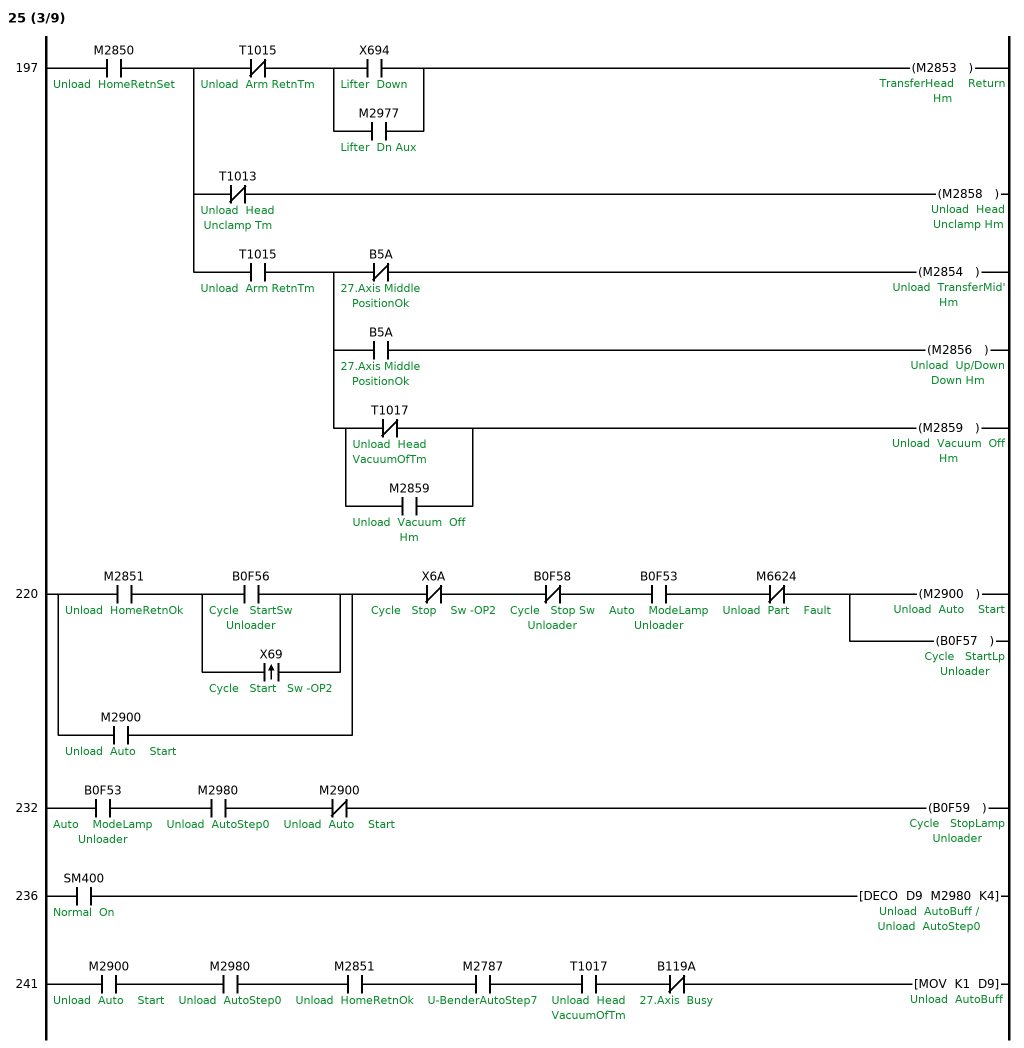
197   LD      M2850  ; Unload  HomeRetnSet
      MPS
      ANI     T1015  ; Unload  Arm RetnTm
      LD      X694  ; Lifter  Down
      OR      M2977  ; Lifter  Dn Aux
      ANB
      OUT     M2853  ; TransferHead    Return  Hm
      MRD
      ANI     T1013  ; Unload  Head    Unclamp Tm
      OUT     M2858  ; Unload  Head    Unclamp Hm
      MPP
      AND     T1015  ; Unload  Arm RetnTm
      MPS
      ANI     B5A  ; 27.Axis Middle  PositionOk
      OUT     M2854  ; Unload  TransferMid' Hm
      MRD
      AND     B5A  ; 27.Axis Middle  PositionOk
      OUT     M2856  ; Unload  Up/Down Down Hm
      MPP
      LDI     T1017  ; Unload  Head    VacuumOfTm
      OR      M2859  ; Unload  Vacuum  Off Hm
      ANB
      OUT     M2859  ; Unload  Vacuum  Off Hm
220   LD      M2851  ; Unload  HomeRetnOk
      LD      B0F56  ; Cycle   StartSw Unloader
      ORP     X69  ; Cycle   Start   Sw -OP2
      ANB
      OR      M2900  ; Unload  Auto    Start
      ANI     X6A  ; Cycle   Stop    Sw -OP2
      ANI     B0F58  ; Cycle   Stop Sw Unloader
      AND     B0F53  ; Auto    ModeLampUnloader
      ANI     M6624  ; Unload  Part    Fault
      OUT     M2900  ; Unload  Auto    Start
      OUT     B0F57  ; Cycle   StartLp Unloader
232   LD      B0F53  ; Auto    ModeLampUnloader
      AND     M2980  ; Unload  AutoStep0
      ANI     M2900  ; Unload  Auto    Start
      OUT     B0F59  ; Cycle   StopLampUnloader
236   LD      SM400  ; Normal  On
      DECO    D9 M2980 K4  ; Unload  AutoBuff
241   LD      M2900  ; Unload  Auto    Start
      AND     M2980  ; Unload  AutoStep0
      AND     M2851  ; Unload  HomeRetnOk
      AND     M2787  ; U-BenderAutoStep7
      AND     T1017  ; Unload  Head    VacuumOfTm
      ANI     B119A  ; 27.Axis  Busy
      MOV     K1 D9
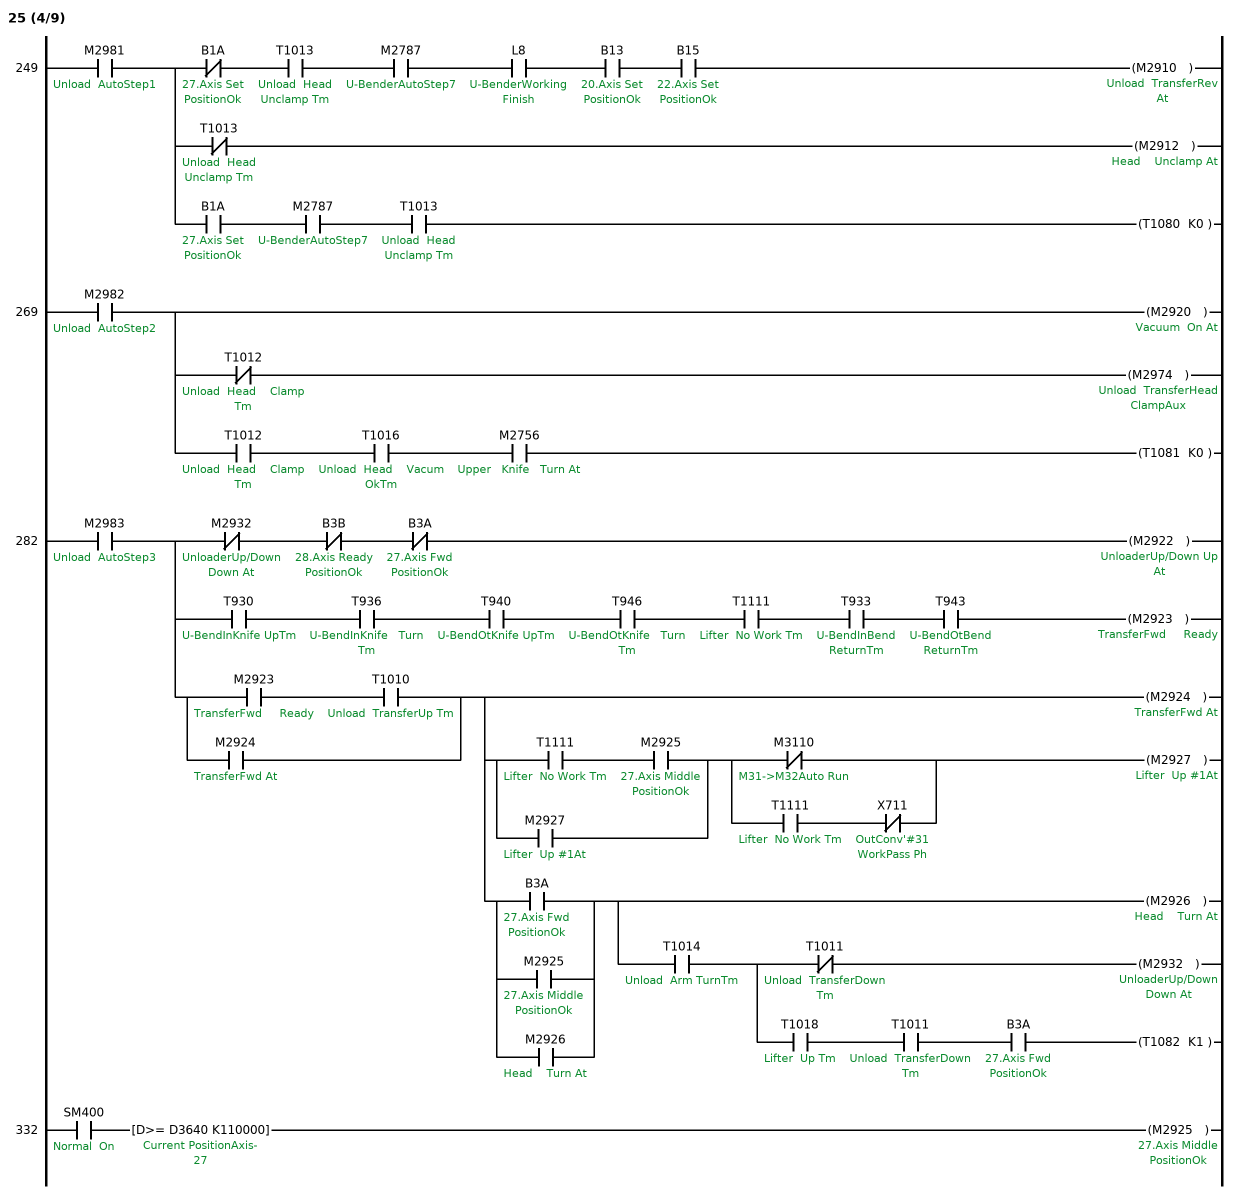
249   LD      M2981  ; Unload  AutoStep1
      MPS
      ANI     B1A  ; 27.Axis Set     PositionOk
      AND     T1013  ; Unload  Head    Unclamp Tm
      AND     M2787  ; U-BenderAutoStep7
      AND     L8  ; U-BenderWorking Finish
      AND     B13  ; 20.Axis Set     PositionOk
      AND     B15  ; 22.Axis Set     PositionOk
      OUT     M2910  ; Unload  TransferRev At
      MRD
      ANI     T1013  ; Unload  Head    Unclamp Tm
      OUT     M2912  ; Head    Unclamp At
      MPP
      AND     B1A  ; 27.Axis Set     PositionOk
      AND     M2787  ; U-BenderAutoStep7
      AND     T1013  ; Unload  Head    Unclamp Tm
      OUT     T1080 K0
269   LD      M2982  ; Unload  AutoStep2
      OUT     M2920  ; Vacuum  On At
      MPS
      ANI     T1012  ; Unload  Head    Clamp Tm
      OUT     M2974  ; Unload  TransferHead    ClampAux
      MPP
      AND     T1012  ; Unload  Head    Clamp Tm
      AND     T1016  ; Unload  Head    Vacum OkTm
      AND     M2756  ; Upper   Knife   Turn At
      OUT     T1081 K0
282   LD      M2983  ; Unload  AutoStep3
      MPS
      ANI     M2932  ; UnloaderUp/Down Down At
      ANI     B3B  ; 28.Axis Ready   PositionOk
      ANI     B3A  ; 27.Axis Fwd     PositionOk
      OUT     M2922  ; UnloaderUp/Down Up At
      MRD
      AND     T930  ; U-BendInKnife UpTm
      AND     T936  ; U-BendInKnife   Turn Tm
      AND     T940  ; U-BendOtKnife UpTm
      AND     T946  ; U-BendOtKnife   Turn Tm
      AND     T1111  ; Lifter  No Work Tm
      AND     T933  ; U-BendInBend    ReturnTm
      AND     T943  ; U-BendOtBend    ReturnTm
      OUT     M2923  ; TransferFwd     Ready
      MPP
      LD      M2923  ; TransferFwd     Ready
      AND     T1010  ; Unload  TransferUp Tm
      OR      M2924  ; TransferFwd At
      ANB
      OUT     M2924  ; TransferFwd At
      MPS
      LD      T1111  ; Lifter  No Work Tm
      AND     M2925  ; 27.Axis Middle  PositionOk
      OR      M2927  ; Lifter  Up #1At
      ANB
      LDI     M3110  ; M31->M32Auto Run
      LD      T1111  ; Lifter  No Work Tm
      ANI     X711  ; OutConv'#31 WorkPass Ph
      ORB
      ANB
      OUT     M2927  ; Lifter  Up #1At
      MPP
      LD      B3A  ; 27.Axis Fwd     PositionOk
      OR      M2925  ; 27.Axis Middle  PositionOk
      OR      M2926  ; Head    Turn At
      ANB
      OUT     M2926  ; Head    Turn At
      AND     T1014  ; Unload  Arm TurnTm
      MPS
      ANI     T1011  ; Unload  TransferDown Tm
      OUT     M2932  ; UnloaderUp/Down Down At
      MPP
      AND     T1018  ; Lifter  Up Tm
      AND     T1011  ; Unload  TransferDown Tm
      AND     B3A  ; 27.Axis Fwd     PositionOk
      OUT     T1082 K1
332   LD      SM400  ; Normal  On
      ANDD>=  D3640 K110000  ; Current PositionAxis-27
      OUT     M2925  ; 27.Axis Middle  PositionOk
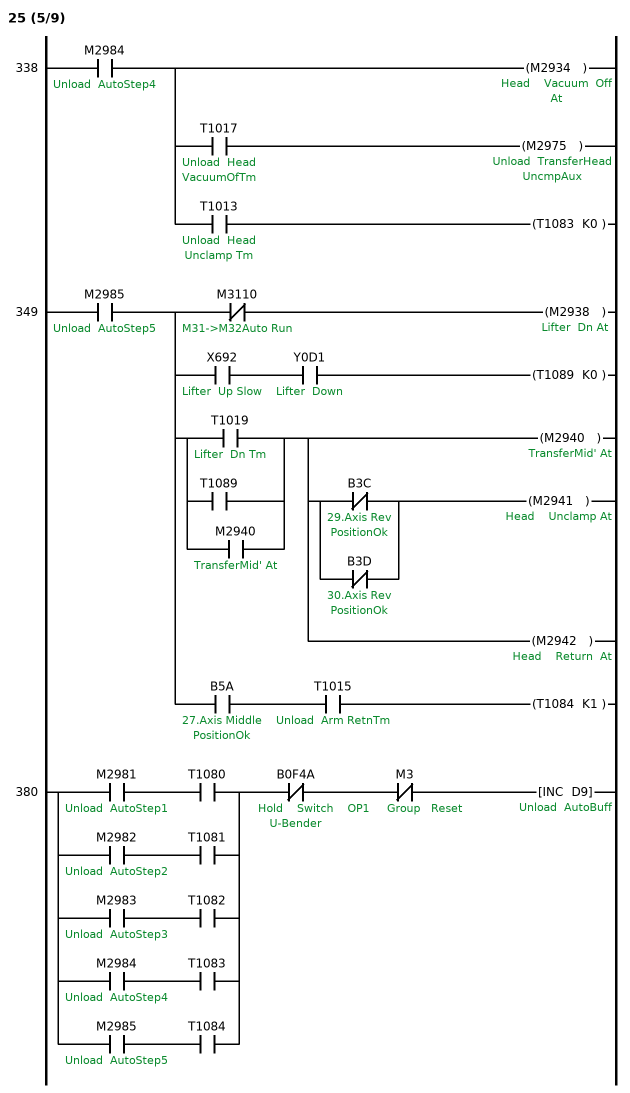
338   LD      M2984  ; Unload  AutoStep4
      OUT     M2934  ; Head    Vacuum  Off At
      MPS
      AND     T1017  ; Unload  Head    VacuumOfTm
      OUT     M2975  ; Unload  TransferHead    UncmpAux
      MPP
      AND     T1013  ; Unload  Head    Unclamp Tm
      OUT     T1083 K0
349   LD      M2985  ; Unload  AutoStep5
      MPS
      ANI     M3110  ; M31->M32Auto Run
      OUT     M2938  ; Lifter  Dn At
      MRD
      AND     X692  ; Lifter  Up Slow
      AND     Y0D1  ; Lifter  Down
      OUT     T1089 K0
      MRD
      LD      T1019  ; Lifter  Dn Tm
      OR      T1089
      OR      M2940  ; TransferMid' At
      ANB
      OUT     M2940  ; TransferMid' At
      MPS
      LDI     B3C  ; 29.Axis Rev     PositionOk
      ORI     B3D  ; 30.Axis Rev     PositionOk
      ANB
      OUT     M2941  ; Head    Unclamp At
      MPP
      OUT     M2942  ; Head    Return  At
      MPP
      AND     B5A  ; 27.Axis Middle  PositionOk
      AND     T1015  ; Unload  Arm RetnTm
      OUT     T1084 K1
380   LD      M2981  ; Unload  AutoStep1
      AND     T1080
      LD      M2982  ; Unload  AutoStep2
      AND     T1081
      ORB
      LD      M2983  ; Unload  AutoStep3
      AND     T1082
      ORB
      LD      M2984  ; Unload  AutoStep4
      AND     T1083
      ORB
      LD      M2985  ; Unload  AutoStep5
      AND     T1084
      ORB
      ANI     B0F4A  ; Hold    Switch  U-Bender
      ANI     M3  ; OP1     Group   Reset
      INC     D9
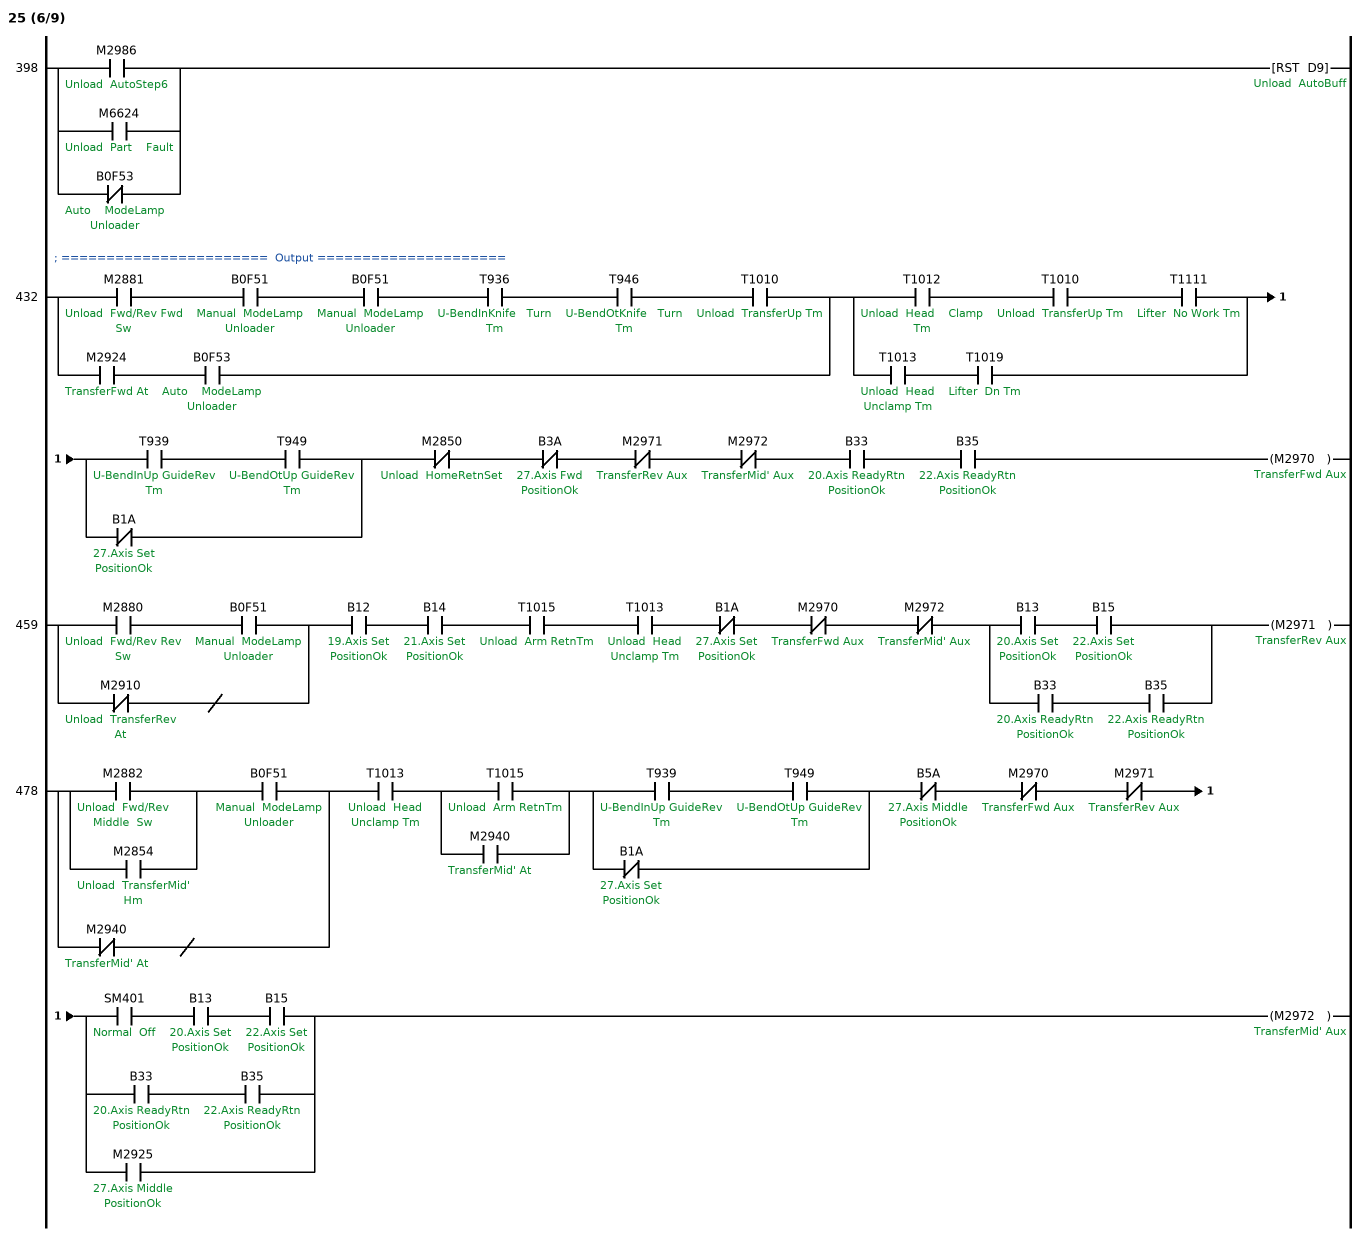
398   LD      M2986  ; Unload  AutoStep6
      OR      M6624  ; Unload  Part    Fault
      ORI     B0F53  ; Auto    ModeLampUnloader
      RST     D9  ; Unload  AutoBuff
; =======================  Output =====================
432   LD      M2881  ; Unload  Fwd/Rev Fwd Sw
      AND     B0F51  ; Manual  ModeLampUnloader
      AND     B0F51  ; Manual  ModeLampUnloader
      AND     T936  ; U-BendInKnife   Turn Tm
      AND     T946  ; U-BendOtKnife   Turn Tm
      AND     T1010  ; Unload  TransferUp Tm
      LD      M2924  ; TransferFwd At
      AND     B0F53  ; Auto    ModeLampUnloader
      ORB
      LD      T1012  ; Unload  Head    Clamp Tm
      AND     T1010  ; Unload  TransferUp Tm
      AND     T1111  ; Lifter  No Work Tm
      LD      T1013  ; Unload  Head    Unclamp Tm
      AND     T1019  ; Lifter  Dn Tm
      ORB
      ANB
      LD      T939  ; U-BendInUp GuideRev Tm
      AND     T949  ; U-BendOtUp GuideRev Tm
      ORI     B1A  ; 27.Axis Set     PositionOk
      ANB
      ANI     M2850  ; Unload  HomeRetnSet
      ANI     B3A  ; 27.Axis Fwd     PositionOk
      ANI     M2971  ; TransferRev Aux
      ANI     M2972  ; TransferMid' Aux
      AND     B33  ; 20.Axis ReadyRtnPositionOk
      AND     B35  ; 22.Axis ReadyRtnPositionOk
      OUT     M2970  ; TransferFwd Aux
459   LD      M2880  ; Unload  Fwd/Rev Rev Sw
      AND     B0F51  ; Manual  ModeLampUnloader
      LDI     M2910  ; Unload  TransferRev At
      INV
      ORB
      AND     B12  ; 19.Axis Set     PositionOk
      AND     B14  ; 21.Axis Set     PositionOk
      AND     T1015  ; Unload  Arm RetnTm
      AND     T1013  ; Unload  Head    Unclamp Tm
      ANI     B1A  ; 27.Axis Set     PositionOk
      ANI     M2970  ; TransferFwd Aux
      ANI     M2972  ; TransferMid' Aux
      LD      B13  ; 20.Axis Set     PositionOk
      AND     B15  ; 22.Axis Set     PositionOk
      LD      B33  ; 20.Axis ReadyRtnPositionOk
      AND     B35  ; 22.Axis ReadyRtnPositionOk
      ORB
      ANB
      OUT     M2971  ; TransferRev Aux
478   LD      M2882  ; Unload  Fwd/Rev Middle  Sw
      OR      M2854  ; Unload  TransferMid' Hm
      AND     B0F51  ; Manual  ModeLampUnloader
      LDI     M2940  ; TransferMid' At
      INV
      ORB
      AND     T1013  ; Unload  Head    Unclamp Tm
      LD      T1015  ; Unload  Arm RetnTm
      OR      M2940  ; TransferMid' At
      ANB
      LD      T939  ; U-BendInUp GuideRev Tm
      AND     T949  ; U-BendOtUp GuideRev Tm
      ORI     B1A  ; 27.Axis Set     PositionOk
      ANB
      ANI     B5A  ; 27.Axis Middle  PositionOk
      ANI     M2970  ; TransferFwd Aux
      ANI     M2971  ; TransferRev Aux
      LD      SM401  ; Normal  Off
      AND     B13  ; 20.Axis Set     PositionOk
      AND     B15  ; 22.Axis Set     PositionOk
      LD      B33  ; 20.Axis ReadyRtnPositionOk
      AND     B35  ; 22.Axis ReadyRtnPositionOk
      ORB
      OR      M2925  ; 27.Axis Middle  PositionOk
      ANB
      OUT     M2972  ; TransferMid' Aux
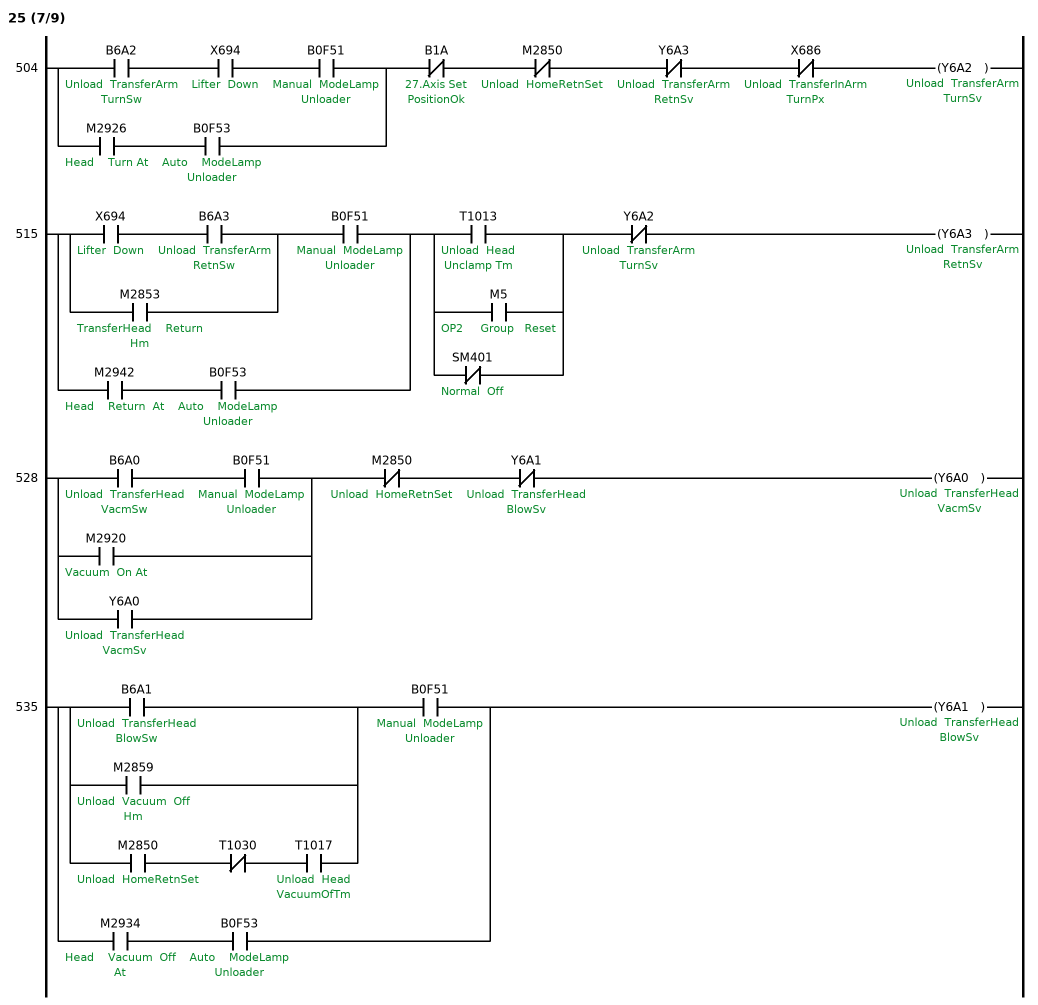
504   LD      B6A2  ; Unload  TransferArm TurnSw
      AND     X694  ; Lifter  Down
      AND     B0F51  ; Manual  ModeLampUnloader
      LD      M2926  ; Head    Turn At
      AND     B0F53  ; Auto    ModeLampUnloader
      ORB
      ANI     B1A  ; 27.Axis Set     PositionOk
      ANI     M2850  ; Unload  HomeRetnSet
      ANI     Y6A3  ; Unload  TransferArm RetnSv
      ANI     X686  ; Unload  TransferInArm   TurnPx
      OUT     Y6A2  ; Unload  TransferArm TurnSv
515   LD      X694  ; Lifter  Down
      AND     B6A3  ; Unload  TransferArm RetnSw
      OR      M2853  ; TransferHead    Return  Hm
      AND     B0F51  ; Manual  ModeLampUnloader
      LD      M2942  ; Head    Return  At
      AND     B0F53  ; Auto    ModeLampUnloader
      ORB
      LD      T1013  ; Unload  Head    Unclamp Tm
      OR      M5  ; OP2     Group   Reset
      ORI     SM401  ; Normal  Off
      ANB
      ANI     Y6A2  ; Unload  TransferArm TurnSv
      OUT     Y6A3  ; Unload  TransferArm RetnSv
528   LD      B6A0  ; Unload  TransferHeadVacmSw
      AND     B0F51  ; Manual  ModeLampUnloader
      OR      M2920  ; Vacuum  On At
      OR      Y6A0  ; Unload  TransferHeadVacmSv
      ANI     M2850  ; Unload  HomeRetnSet
      ANI     Y6A1  ; Unload  TransferHeadBlowSv
      OUT     Y6A0  ; Unload  TransferHeadVacmSv
535   LD      B6A1  ; Unload  TransferHeadBlowSw
      OR      M2859  ; Unload  Vacuum  Off Hm
      LD      M2850  ; Unload  HomeRetnSet
      ANI     T1030
      AND     T1017  ; Unload  Head    VacuumOfTm
      ORB
      AND     B0F51  ; Manual  ModeLampUnloader
      LD      M2934  ; Head    Vacuum  Off At
      AND     B0F53  ; Auto    ModeLampUnloader
      ORB
      OUT     Y6A1  ; Unload  TransferHeadBlowSv
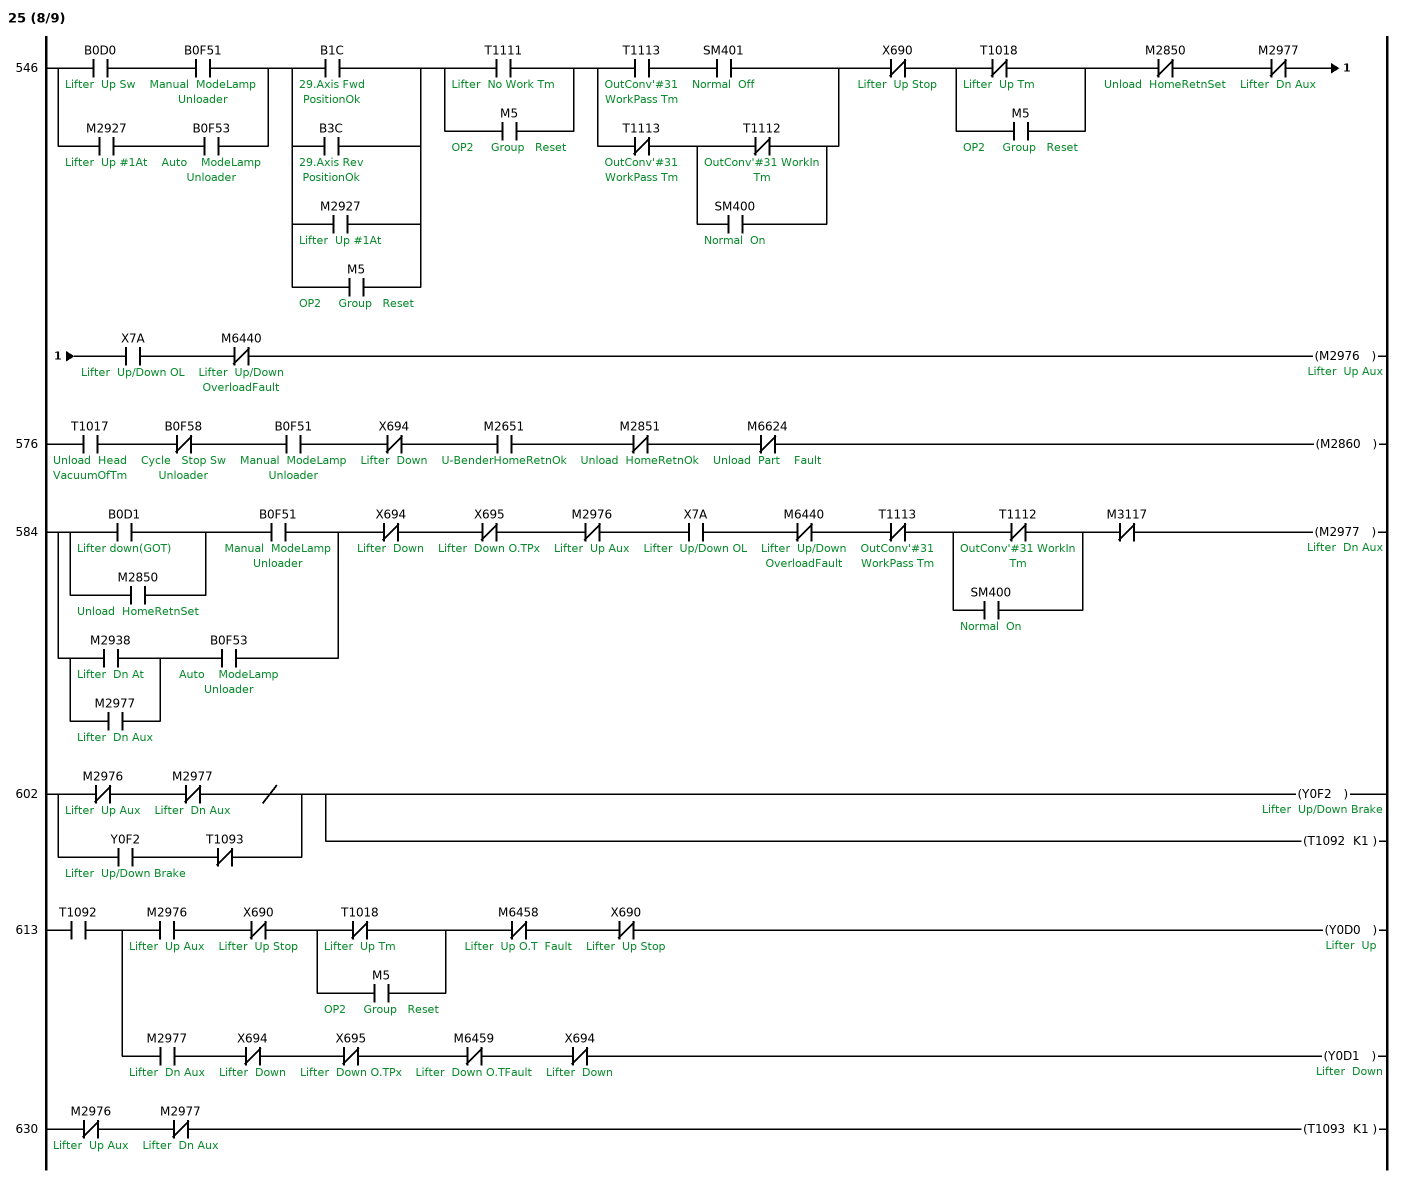
546   LD      B0D0  ; Lifter  Up Sw
      AND     B0F51  ; Manual  ModeLampUnloader
      LD      M2927  ; Lifter  Up #1At
      AND     B0F53  ; Auto    ModeLampUnloader
      ORB
      LD      B1C  ; 29.Axis Fwd     PositionOk
      OR      B3C  ; 29.Axis Rev     PositionOk
      OR      M2927  ; Lifter  Up #1At
      OR      M5  ; OP2     Group   Reset
      ANB
      LD      T1111  ; Lifter  No Work Tm
      OR      M5  ; OP2     Group   Reset
      ANB
      LD      T1113  ; OutConv'#31 WorkPass Tm
      AND     SM401  ; Normal  Off
      LDI     T1113  ; OutConv'#31 WorkPass Tm
      LDI     T1112  ; OutConv'#31 WorkIn  Tm
      OR      SM400  ; Normal  On
      ANB
      ORB
      ANB
      ANI     X690  ; Lifter  Up Stop
      LDI     T1018  ; Lifter  Up Tm
      OR      M5  ; OP2     Group   Reset
      ANB
      ANI     M2850  ; Unload  HomeRetnSet
      ANI     M2977  ; Lifter  Dn Aux
      AND     X7A  ; Lifter  Up/Down OL
      ANI     M6440  ; Lifter  Up/Down OverloadFault
      OUT     M2976  ; Lifter  Up Aux
576   LD      T1017  ; Unload  Head    VacuumOfTm
      ANI     B0F58  ; Cycle   Stop Sw Unloader
      AND     B0F51  ; Manual  ModeLampUnloader
      ANI     X694  ; Lifter  Down
      AND     M2651  ; U-BenderHomeRetnOk
      ANI     M2851  ; Unload  HomeRetnOk
      ANI     M6624  ; Unload  Part    Fault
      OUT     M2860
584   LD      B0D1  ; Lifter down(GOT)
      OR      M2850  ; Unload  HomeRetnSet
      AND     B0F51  ; Manual  ModeLampUnloader
      LD      M2938  ; Lifter  Dn At
      OR      M2977  ; Lifter  Dn Aux
      AND     B0F53  ; Auto    ModeLampUnloader
      ORB
      ANI     X694  ; Lifter  Down
      ANI     X695  ; Lifter  Down O.TPx
      ANI     M2976  ; Lifter  Up Aux
      AND     X7A  ; Lifter  Up/Down OL
      ANI     M6440  ; Lifter  Up/Down OverloadFault
      ANI     T1113  ; OutConv'#31 WorkPass Tm
      LDI     T1112  ; OutConv'#31 WorkIn  Tm
      OR      SM400  ; Normal  On
      ANB
      ANI     M3117
      OUT     M2977  ; Lifter  Dn Aux
602   LDI     M2976  ; Lifter  Up Aux
      ANI     M2977  ; Lifter  Dn Aux
      INV
      LD      Y0F2  ; Lifter  Up/Down Brake
      ANI     T1093
      ORB
      OUT     Y0F2  ; Lifter  Up/Down Brake
      OUT     T1092 K1
613   LD      T1092
      MPS
      AND     M2976  ; Lifter  Up Aux
      ANI     X690  ; Lifter  Up Stop
      LDI     T1018  ; Lifter  Up Tm
      OR      M5  ; OP2     Group   Reset
      ANB
      ANI     M6458  ; Lifter  Up O.T  Fault
      ANI     X690  ; Lifter  Up Stop
      OUT     Y0D0  ; Lifter  Up
      MPP
      AND     M2977  ; Lifter  Dn Aux
      ANI     X694  ; Lifter  Down
      ANI     X695  ; Lifter  Down O.TPx
      ANI     M6459  ; Lifter  Down O.TFault
      ANI     X694  ; Lifter  Down
      OUT     Y0D1  ; Lifter  Down
630   LDI     M2976  ; Lifter  Up Aux
      ANI     M2977  ; Lifter  Dn Aux
      OUT     T1093 K1
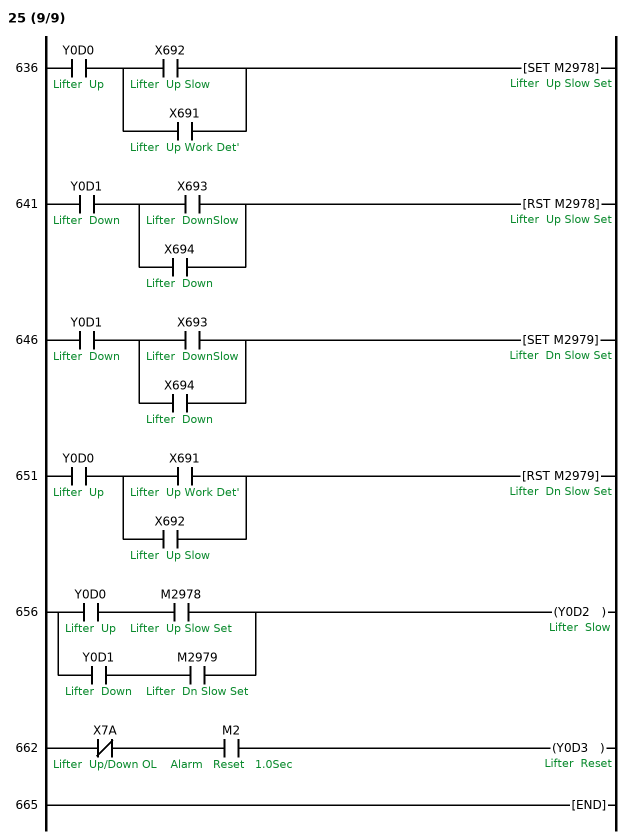
636   LD      Y0D0  ; Lifter  Up
      LD      X692  ; Lifter  Up Slow
      OR      X691  ; Lifter  Up Work Det'
      ANB
      SET     M2978  ; Lifter  Up Slow Set
641   LD      Y0D1  ; Lifter  Down
      LD      X693  ; Lifter  DownSlow
      OR      X694  ; Lifter  Down
      ANB
      RST     M2978  ; Lifter  Up Slow Set
646   LD      Y0D1  ; Lifter  Down
      LD      X693  ; Lifter  DownSlow
      OR      X694  ; Lifter  Down
      ANB
      SET     M2979  ; Lifter  Dn Slow Set
651   LD      Y0D0  ; Lifter  Up
      LD      X691  ; Lifter  Up Work Det'
      OR      X692  ; Lifter  Up Slow
      ANB
      RST     M2979  ; Lifter  Dn Slow Set
656   LD      Y0D0  ; Lifter  Up
      AND     M2978  ; Lifter  Up Slow Set
      LD      Y0D1  ; Lifter  Down
      AND     M2979  ; Lifter  Dn Slow Set
      ORB
      OUT     Y0D2  ; Lifter  Slow
662   LDI     X7A  ; Lifter  Up/Down OL
      AND     M2  ; Alarm   Reset   1.0Sec
      OUT     Y0D3  ; Lifter  Reset
665   END
END_PROGRAM

PROGRAM 26  // Out Conveyor
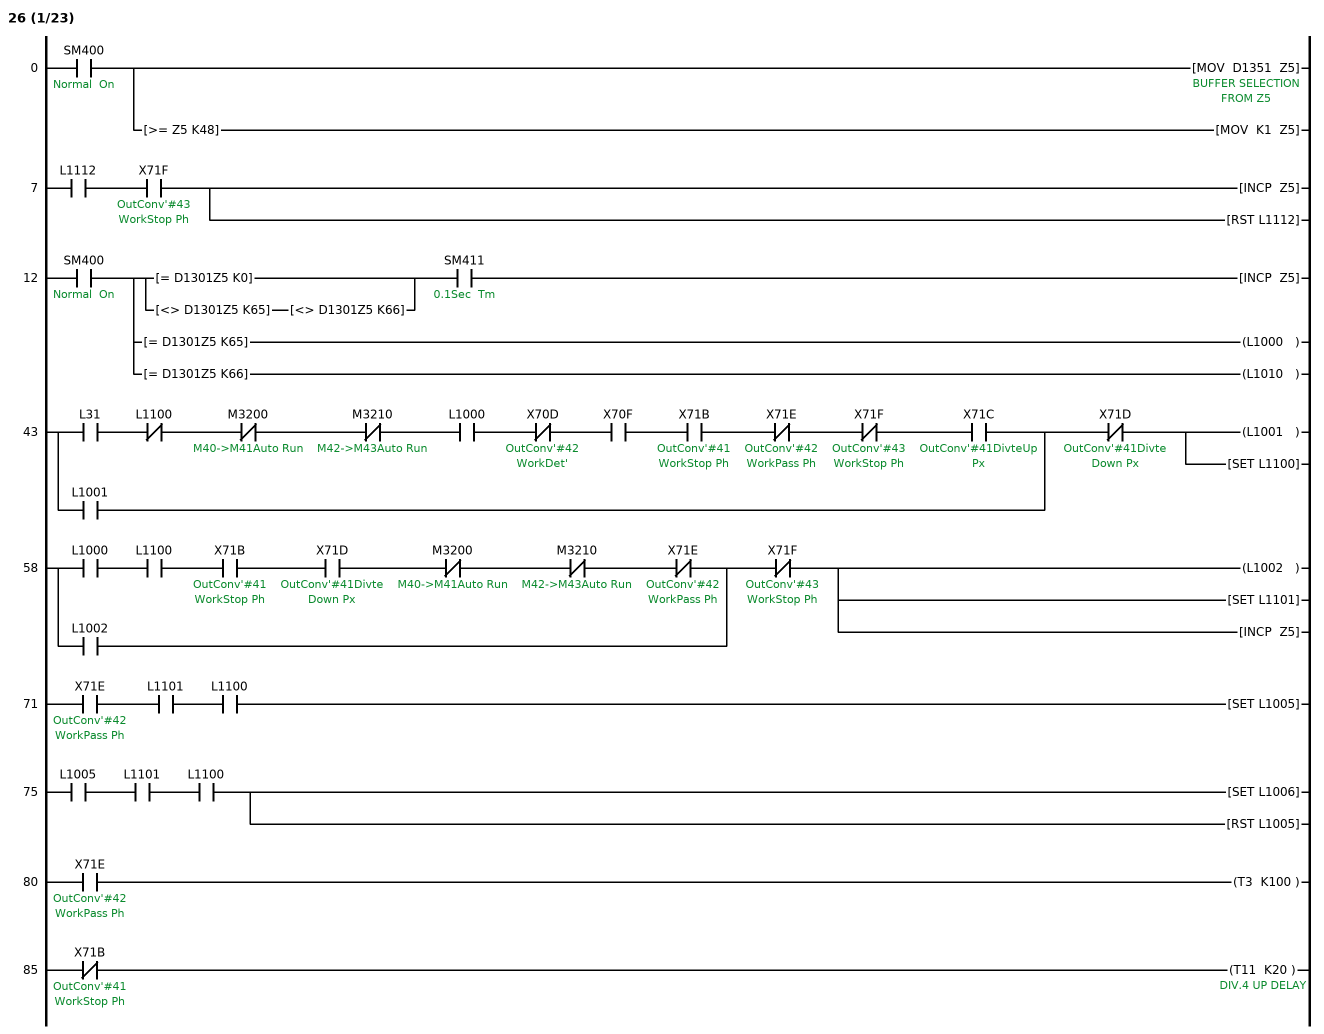
0     LD      SM400  ; Normal  On
      MOV     D1351 Z5  ; BUFFER SELECTION FROM Z5
      AND>=   Z5 K48
      MOV     K1 Z5
7     LD      L1112
      AND     X71F  ; OutConv'#43 WorkStop Ph
      INCP    Z5
      RST     L1112
12    LD      SM400  ; Normal  On
      MPS
      LD=     D1301Z5 K0
      LD<>    D1301Z5 K65
      AND<>   D1301Z5 K66
      ORB
      ANB
      AND     SM411  ; 0.1Sec  Tm
      INCP    Z5
      MRD
      AND=    D1301Z5 K65
      OUT     L1000
      MPP
      AND=    D1301Z5 K66
      OUT     L1010
43    LD      L31
      ANI     L1100
      ANI     M3200  ; M40->M41Auto Run
      ANI     M3210  ; M42->M43Auto Run
      AND     L1000
      ANI     X70D  ; OutConv'#42 WorkDet'
      AND     X70F
      AND     X71B  ; OutConv'#41 WorkStop Ph
      ANI     X71E  ; OutConv'#42 WorkPass Ph
      ANI     X71F  ; OutConv'#43 WorkStop Ph
      AND     X71C  ; OutConv'#41DivteUp Px
      OR      L1001
      ANI     X71D  ; OutConv'#41DivteDown Px
      OUT     L1001
      SET     L1100
58    LD      L1000
      AND     L1100
      AND     X71B  ; OutConv'#41 WorkStop Ph
      AND     X71D  ; OutConv'#41DivteDown Px
      ANI     M3200  ; M40->M41Auto Run
      ANI     M3210  ; M42->M43Auto Run
      ANI     X71E  ; OutConv'#42 WorkPass Ph
      OR      L1002
      ANI     X71F  ; OutConv'#43 WorkStop Ph
      OUT     L1002
      SET     L1101
      INCP    Z5
71    LD      X71E  ; OutConv'#42 WorkPass Ph
      AND     L1101
      AND     L1100
      SET     L1005
75    LD      L1005
      AND     L1101
      AND     L1100
      SET     L1006
      RST     L1005
80    LD      X71E  ; OutConv'#42 WorkPass Ph
      OUT     T3 K100
85    LDI     X71B  ; OutConv'#41 WorkStop Ph
      OUT     T11 K20  ; DIV.4 UP DELAY
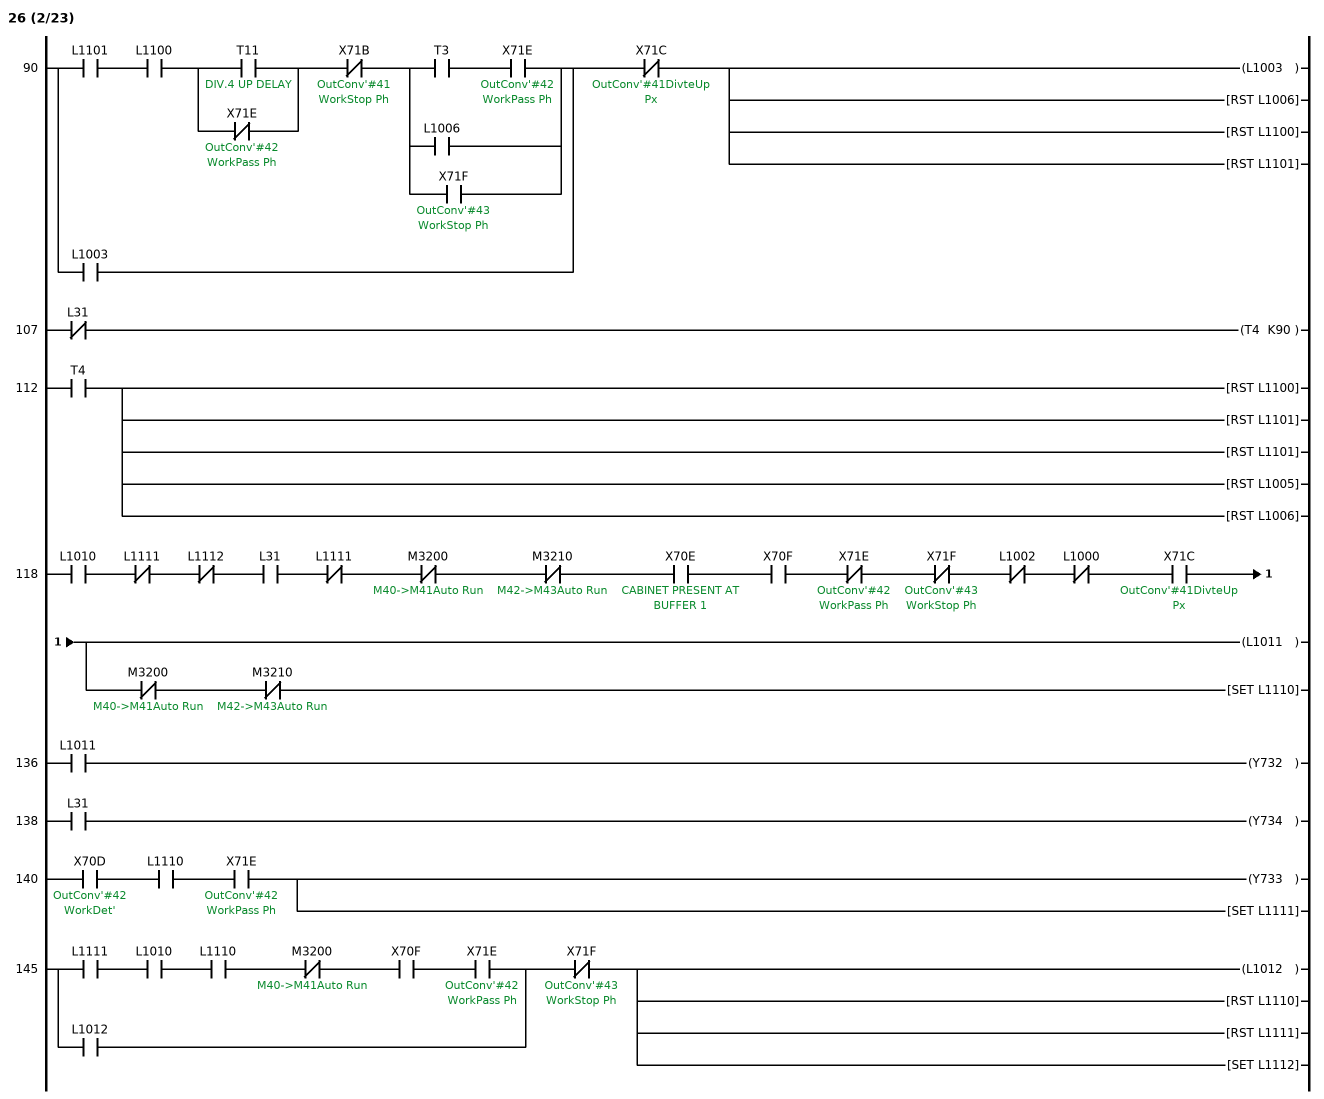
90    LD      L1101
      AND     L1100
      LD      T11  ; DIV.4 UP DELAY
      ORI     X71E  ; OutConv'#42 WorkPass Ph
      ANB
      ANI     X71B  ; OutConv'#41 WorkStop Ph
      LD      T3
      AND     X71E  ; OutConv'#42 WorkPass Ph
      OR      L1006
      OR      X71F  ; OutConv'#43 WorkStop Ph
      ANB
      OR      L1003
      ANI     X71C  ; OutConv'#41DivteUp Px
      OUT     L1003
      RST     L1006
      RST     L1100
      RST     L1101
107   LDI     L31
      OUT     T4 K90
112   LD      T4
      RST     L1100
      RST     L1101
      RST     L1101
      RST     L1005
      RST     L1006
118   LD      L1010
      ANI     L1111
      ANI     L1112
      AND     L31
      ANI     L1111
      ANI     M3200  ; M40->M41Auto Run
      ANI     M3210  ; M42->M43Auto Run
      AND     X70E  ; CABINET PRESENT AT BUFFER 1
      AND     X70F
      ANI     X71E  ; OutConv'#42 WorkPass Ph
      ANI     X71F  ; OutConv'#43 WorkStop Ph
      ANI     L1002
      ANI     L1000
      AND     X71C  ; OutConv'#41DivteUp Px
      OUT     L1011
      ANI     M3200  ; M40->M41Auto Run
      ANI     M3210  ; M42->M43Auto Run
      SET     L1110
136   LD      L1011
      OUT     Y732
138   LD      L31
      OUT     Y734
140   LD      X70D  ; OutConv'#42 WorkDet'
      AND     L1110
      AND     X71E  ; OutConv'#42 WorkPass Ph
      OUT     Y733
      SET     L1111
145   LD      L1111
      AND     L1010
      AND     L1110
      ANI     M3200  ; M40->M41Auto Run
      AND     X70F
      AND     X71E  ; OutConv'#42 WorkPass Ph
      OR      L1012
      ANI     X71F  ; OutConv'#43 WorkStop Ph
      OUT     L1012
      RST     L1110
      RST     L1111
      SET     L1112
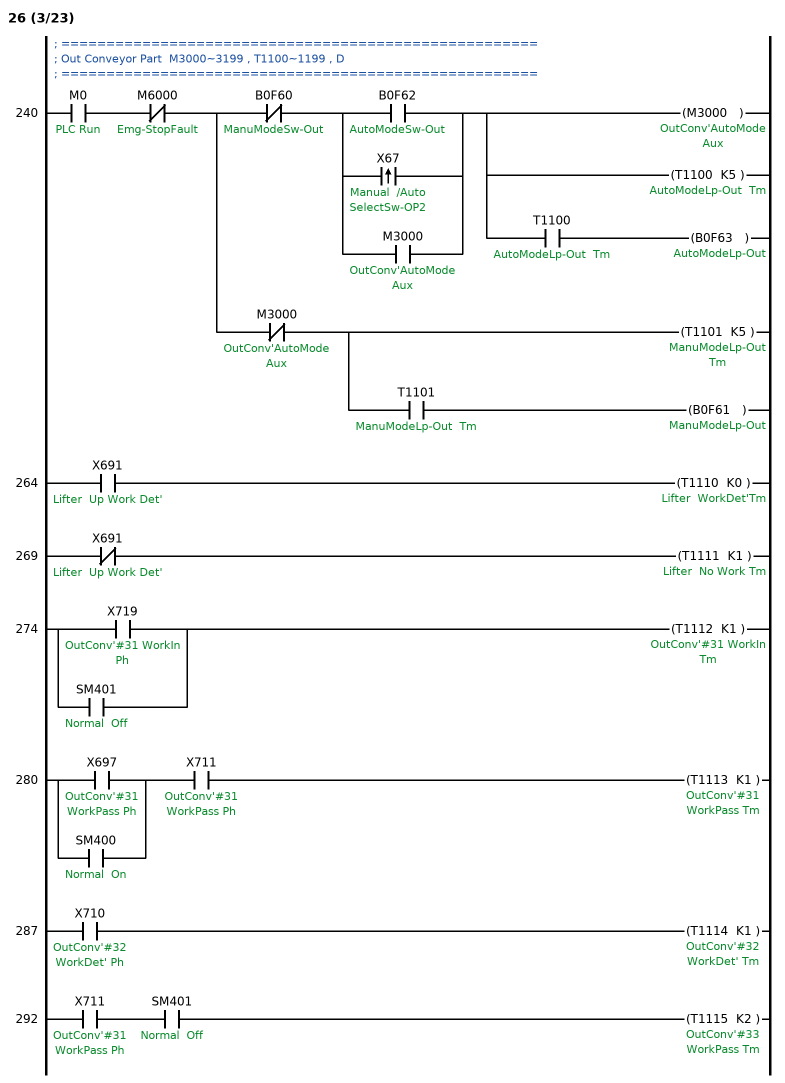
; =====================================================
; Out Conveyor Part  M3000~3199 , T1100~1199 , D
; =====================================================
240   LD      M0  ; PLC Run
      ANI     M6000  ; Emg-StopFault
      MPS
      ANI     B0F60  ; ManuModeSw-Out
      LD      B0F62  ; AutoModeSw-Out
      ORP     X67  ; Manual  /Auto   SelectSw-OP2
      OR      M3000  ; OutConv'AutoModeAux
      ANB
      OUT     M3000  ; OutConv'AutoModeAux
      OUT     T1100 K5  ; AutoModeLp-Out  Tm
      AND     T1100  ; AutoModeLp-Out  Tm
      OUT     B0F63  ; AutoModeLp-Out
      MPP
      ANI     M3000  ; OutConv'AutoModeAux
      OUT     T1101 K5  ; ManuModeLp-Out  Tm
      AND     T1101  ; ManuModeLp-Out  Tm
      OUT     B0F61  ; ManuModeLp-Out
264   LD      X691  ; Lifter  Up Work Det'
      OUT     T1110 K0  ; Lifter  WorkDet'Tm
269   LDI     X691  ; Lifter  Up Work Det'
      OUT     T1111 K1  ; Lifter  No Work Tm
274   LD      X719  ; OutConv'#31 WorkIn  Ph
      OR      SM401  ; Normal  Off
      OUT     T1112 K1  ; OutConv'#31 WorkIn  Tm
280   LD      X697  ; OutConv'#31 WorkPass Ph
      OR      SM400  ; Normal  On
      AND     X711  ; OutConv'#31 WorkPass Ph
      OUT     T1113 K1  ; OutConv'#31 WorkPass Tm
287   LD      X710  ; OutConv'#32 WorkDet' Ph
      OUT     T1114 K1  ; OutConv'#32 WorkDet' Tm
292   LD      X711  ; OutConv'#31 WorkPass Ph
      AND     SM401  ; Normal  Off
      OUT     T1115 K2  ; OutConv'#33 WorkPass Tm
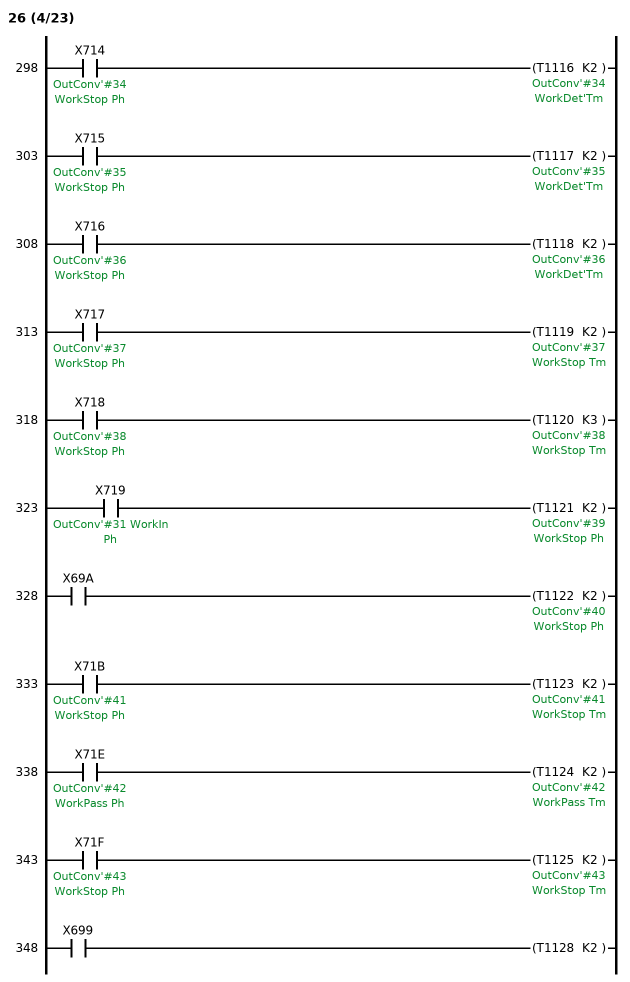
298   LD      X714  ; OutConv'#34 WorkStop Ph
      OUT     T1116 K2  ; OutConv'#34 WorkDet'Tm
303   LD      X715  ; OutConv'#35 WorkStop Ph
      OUT     T1117 K2  ; OutConv'#35 WorkDet'Tm
308   LD      X716  ; OutConv'#36 WorkStop Ph
      OUT     T1118 K2  ; OutConv'#36 WorkDet'Tm
313   LD      X717  ; OutConv'#37 WorkStop Ph
      OUT     T1119 K2  ; OutConv'#37 WorkStop Tm
318   LD      X718  ; OutConv'#38 WorkStop Ph
      OUT     T1120 K3  ; OutConv'#38 WorkStop Tm
323   LD      X719  ; OutConv'#31 WorkIn  Ph
      OUT     T1121 K2  ; OutConv'#39 WorkStop Ph
328   LD      X69A
      OUT     T1122 K2  ; OutConv'#40 WorkStop Ph
333   LD      X71B  ; OutConv'#41 WorkStop Ph
      OUT     T1123 K2  ; OutConv'#41 WorkStop Tm
338   LD      X71E  ; OutConv'#42 WorkPass Ph
      OUT     T1124 K2  ; OutConv'#42 WorkPass Tm
343   LD      X71F  ; OutConv'#43 WorkStop Ph
      OUT     T1125 K2  ; OutConv'#43 WorkStop Tm
348   LD      X699
      OUT     T1128 K2
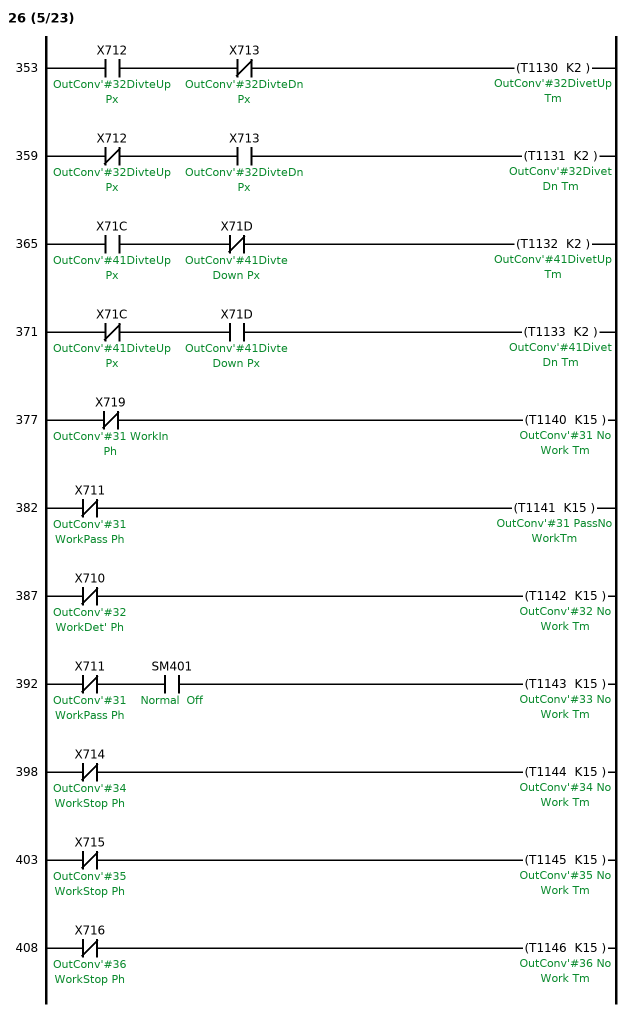
353   LD      X712  ; OutConv'#32DivteUp Px
      ANI     X713  ; OutConv'#32DivteDn Px
      OUT     T1130 K2  ; OutConv'#32DivetUp Tm
359   LDI     X712  ; OutConv'#32DivteUp Px
      AND     X713  ; OutConv'#32DivteDn Px
      OUT     T1131 K2  ; OutConv'#32DivetDn Tm
365   LD      X71C  ; OutConv'#41DivteUp Px
      ANI     X71D  ; OutConv'#41DivteDown Px
      OUT     T1132 K2  ; OutConv'#41DivetUp Tm
371   LDI     X71C  ; OutConv'#41DivteUp Px
      AND     X71D  ; OutConv'#41DivteDown Px
      OUT     T1133 K2  ; OutConv'#41DivetDn Tm
377   LDI     X719  ; OutConv'#31 WorkIn  Ph
      OUT     T1140 K15  ; OutConv'#31 No  Work Tm
382   LDI     X711  ; OutConv'#31 WorkPass Ph
      OUT     T1141 K15  ; OutConv'#31 PassNo  WorkTm
387   LDI     X710  ; OutConv'#32 WorkDet' Ph
      OUT     T1142 K15  ; OutConv'#32 No  Work Tm
392   LDI     X711  ; OutConv'#31 WorkPass Ph
      AND     SM401  ; Normal  Off
      OUT     T1143 K15  ; OutConv'#33 No  Work Tm
398   LDI     X714  ; OutConv'#34 WorkStop Ph
      OUT     T1144 K15  ; OutConv'#34 No  Work Tm
403   LDI     X715  ; OutConv'#35 WorkStop Ph
      OUT     T1145 K15  ; OutConv'#35 No  Work Tm
408   LDI     X716  ; OutConv'#36 WorkStop Ph
      OUT     T1146 K15  ; OutConv'#36 No  Work Tm
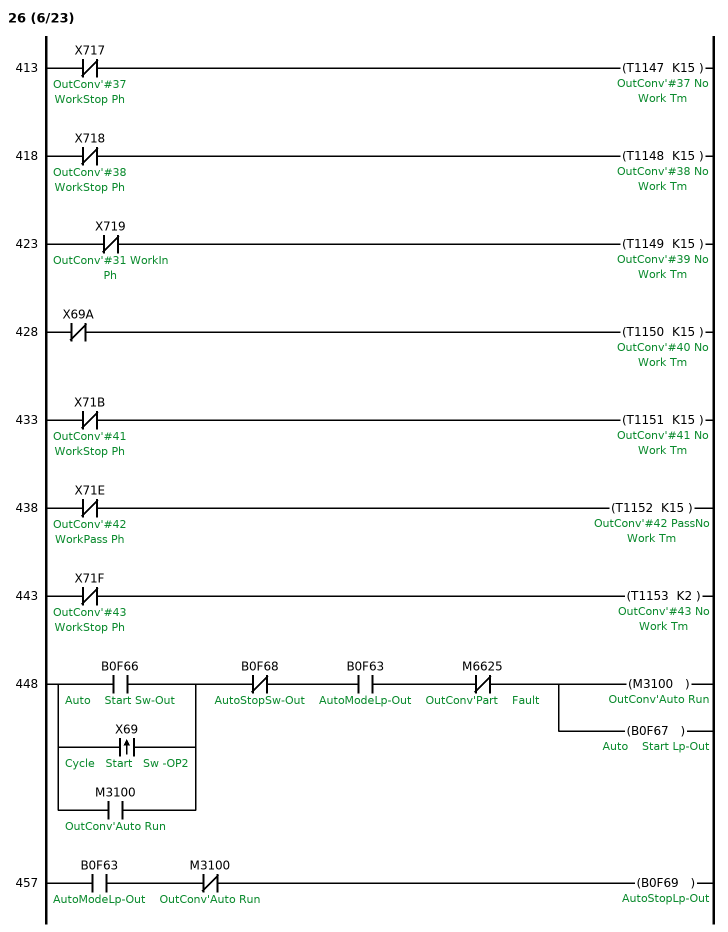
413   LDI     X717  ; OutConv'#37 WorkStop Ph
      OUT     T1147 K15  ; OutConv'#37 No  Work Tm
418   LDI     X718  ; OutConv'#38 WorkStop Ph
      OUT     T1148 K15  ; OutConv'#38 No  Work Tm
423   LDI     X719  ; OutConv'#31 WorkIn  Ph
      OUT     T1149 K15  ; OutConv'#39 No  Work Tm
428   LDI     X69A
      OUT     T1150 K15  ; OutConv'#40 No  Work Tm
433   LDI     X71B  ; OutConv'#41 WorkStop Ph
      OUT     T1151 K15  ; OutConv'#41 No  Work Tm
438   LDI     X71E  ; OutConv'#42 WorkPass Ph
      OUT     T1152 K15  ; OutConv'#42 PassNo Work Tm
443   LDI     X71F  ; OutConv'#43 WorkStop Ph
      OUT     T1153 K2  ; OutConv'#43 No  Work Tm
448   LD      B0F66  ; Auto    Start Sw-Out
      ORP     X69  ; Cycle   Start   Sw -OP2
      OR      M3100  ; OutConv'Auto Run
      ANI     B0F68  ; AutoStopSw-Out
      AND     B0F63  ; AutoModeLp-Out
      ANI     M6625  ; OutConv'Part    Fault
      OUT     M3100  ; OutConv'Auto Run
      OUT     B0F67  ; Auto    Start Lp-Out
457   LD      B0F63  ; AutoModeLp-Out
      ANI     M3100  ; OutConv'Auto Run
      OUT     B0F69  ; AutoStopLp-Out
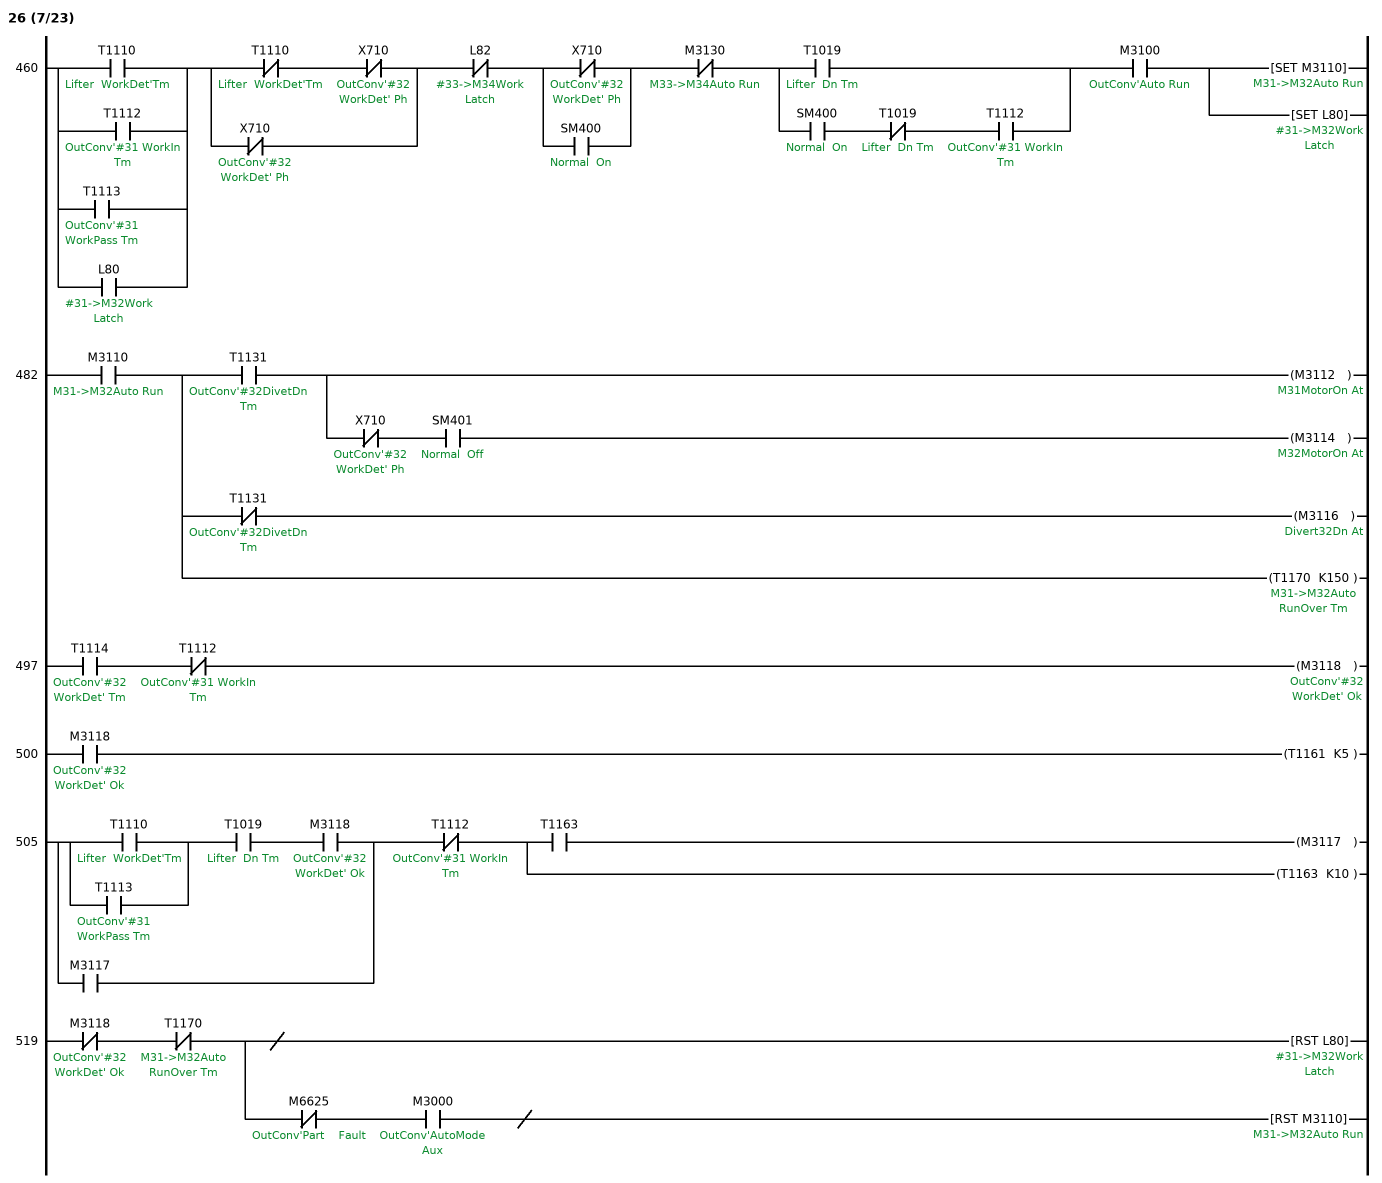
460   LD      T1110  ; Lifter  WorkDet'Tm
      OR      T1112  ; OutConv'#31 WorkIn  Tm
      OR      T1113  ; OutConv'#31 WorkPass Tm
      OR      L80  ; #31->M32Work    Latch
      LDI     T1110  ; Lifter  WorkDet'Tm
      ANI     X710  ; OutConv'#32 WorkDet' Ph
      ORI     X710  ; OutConv'#32 WorkDet' Ph
      ANB
      ANI     L82  ; #33->M34Work    Latch
      LDI     X710  ; OutConv'#32 WorkDet' Ph
      OR      SM400  ; Normal  On
      ANB
      ANI     M3130  ; M33->M34Auto Run
      LD      T1019  ; Lifter  Dn Tm
      LD      SM400  ; Normal  On
      ANI     T1019  ; Lifter  Dn Tm
      AND     T1112  ; OutConv'#31 WorkIn  Tm
      ORB
      ANB
      AND     M3100  ; OutConv'Auto Run
      SET     M3110  ; M31->M32Auto Run
      SET     L80  ; #31->M32Work    Latch
482   LD      M3110  ; M31->M32Auto Run
      MPS
      AND     T1131  ; OutConv'#32DivetDn Tm
      OUT     M3112  ; M31MotorOn At
      ANI     X710  ; OutConv'#32 WorkDet' Ph
      AND     SM401  ; Normal  Off
      OUT     M3114  ; M32MotorOn At
      MRD
      ANI     T1131  ; OutConv'#32DivetDn Tm
      OUT     M3116  ; Divert32Dn At
      MPP
      OUT     T1170 K150  ; M31->M32Auto RunOver Tm
497   LD      T1114  ; OutConv'#32 WorkDet' Tm
      ANI     T1112  ; OutConv'#31 WorkIn  Tm
      OUT     M3118  ; OutConv'#32 WorkDet' Ok
500   LD      M3118  ; OutConv'#32 WorkDet' Ok
      OUT     T1161 K5
505   LD      T1110  ; Lifter  WorkDet'Tm
      OR      T1113  ; OutConv'#31 WorkPass Tm
      AND     T1019  ; Lifter  Dn Tm
      AND     M3118  ; OutConv'#32 WorkDet' Ok
      OR      M3117
      ANI     T1112  ; OutConv'#31 WorkIn  Tm
      MPS
      AND     T1163
      OUT     M3117
      MPP
      OUT     T1163 K10
519   LDI     M3118  ; OutConv'#32 WorkDet' Ok
      ANI     T1170  ; M31->M32Auto RunOver Tm
      MPS
      INV
      RST     L80  ; #31->M32Work    Latch
      MPP
      ANI     M6625  ; OutConv'Part    Fault
      AND     M3000  ; OutConv'AutoModeAux
      INV
      RST     M3110  ; M31->M32Auto Run
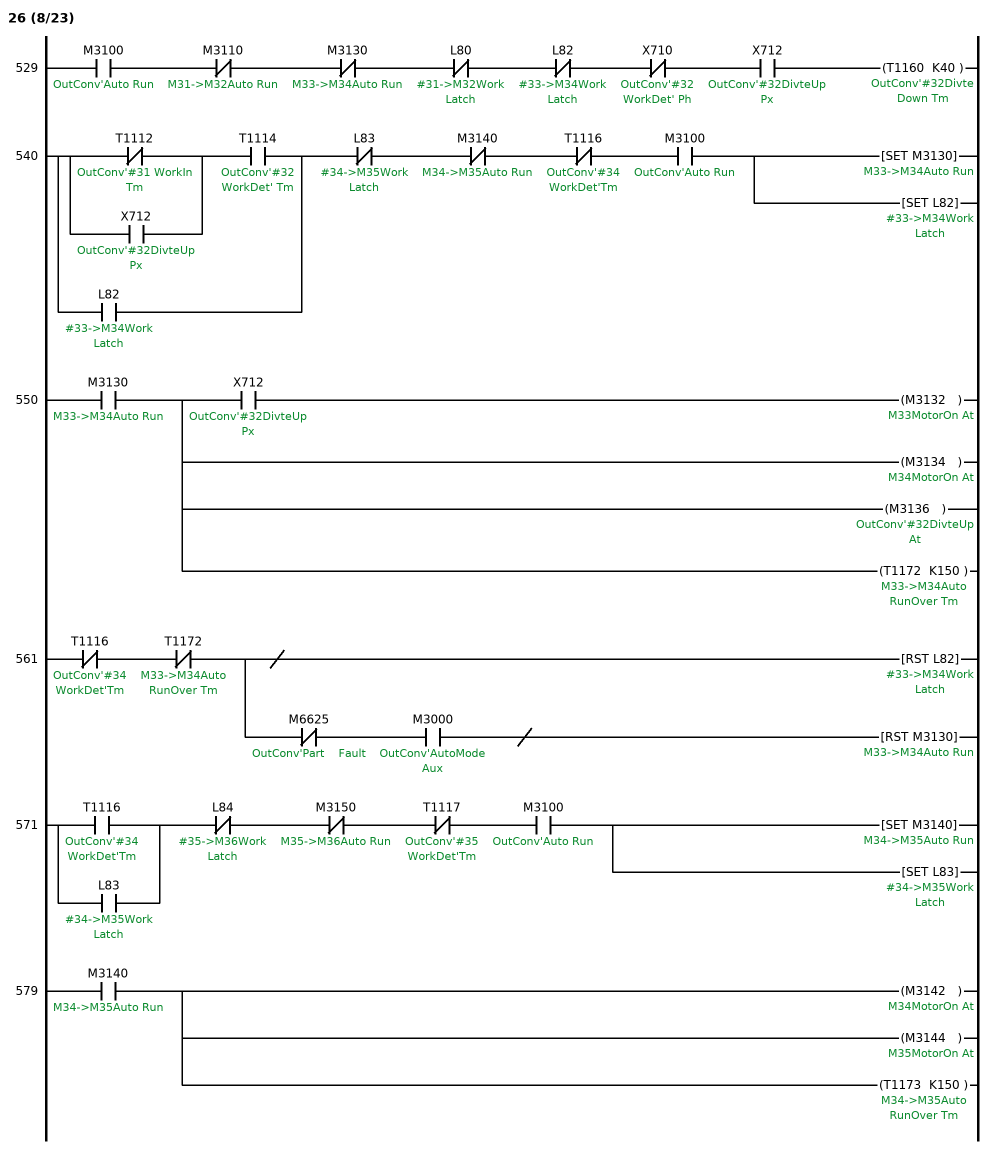
529   LD      M3100  ; OutConv'Auto Run
      ANI     M3110  ; M31->M32Auto Run
      ANI     M3130  ; M33->M34Auto Run
      ANI     L80  ; #31->M32Work    Latch
      ANI     L82  ; #33->M34Work    Latch
      ANI     X710  ; OutConv'#32 WorkDet' Ph
      AND     X712  ; OutConv'#32DivteUp Px
      OUT     T1160 K40  ; OutConv'#32DivteDown Tm
540   LDI     T1112  ; OutConv'#31 WorkIn  Tm
      OR      X712  ; OutConv'#32DivteUp Px
      AND     T1114  ; OutConv'#32 WorkDet' Tm
      OR      L82  ; #33->M34Work    Latch
      ANI     L83  ; #34->M35Work    Latch
      ANI     M3140  ; M34->M35Auto Run
      ANI     T1116  ; OutConv'#34 WorkDet'Tm
      AND     M3100  ; OutConv'Auto Run
      SET     M3130  ; M33->M34Auto Run
      SET     L82  ; #33->M34Work    Latch
550   LD      M3130  ; M33->M34Auto Run
      MPS
      AND     X712  ; OutConv'#32DivteUp Px
      OUT     M3132  ; M33MotorOn At
      MPP
      OUT     M3134  ; M34MotorOn At
      OUT     M3136  ; OutConv'#32DivteUp At
      OUT     T1172 K150  ; M33->M34Auto RunOver Tm
561   LDI     T1116  ; OutConv'#34 WorkDet'Tm
      ANI     T1172  ; M33->M34Auto RunOver Tm
      MPS
      INV
      RST     L82  ; #33->M34Work    Latch
      MPP
      ANI     M6625  ; OutConv'Part    Fault
      AND     M3000  ; OutConv'AutoModeAux
      INV
      RST     M3130  ; M33->M34Auto Run
571   LD      T1116  ; OutConv'#34 WorkDet'Tm
      OR      L83  ; #34->M35Work    Latch
      ANI     L84  ; #35->M36Work    Latch
      ANI     M3150  ; M35->M36Auto Run
      ANI     T1117  ; OutConv'#35 WorkDet'Tm
      AND     M3100  ; OutConv'Auto Run
      SET     M3140  ; M34->M35Auto Run
      SET     L83  ; #34->M35Work    Latch
579   LD      M3140  ; M34->M35Auto Run
      OUT     M3142  ; M34MotorOn At
      OUT     M3144  ; M35MotorOn At
      OUT     T1173 K150  ; M34->M35Auto RunOver Tm
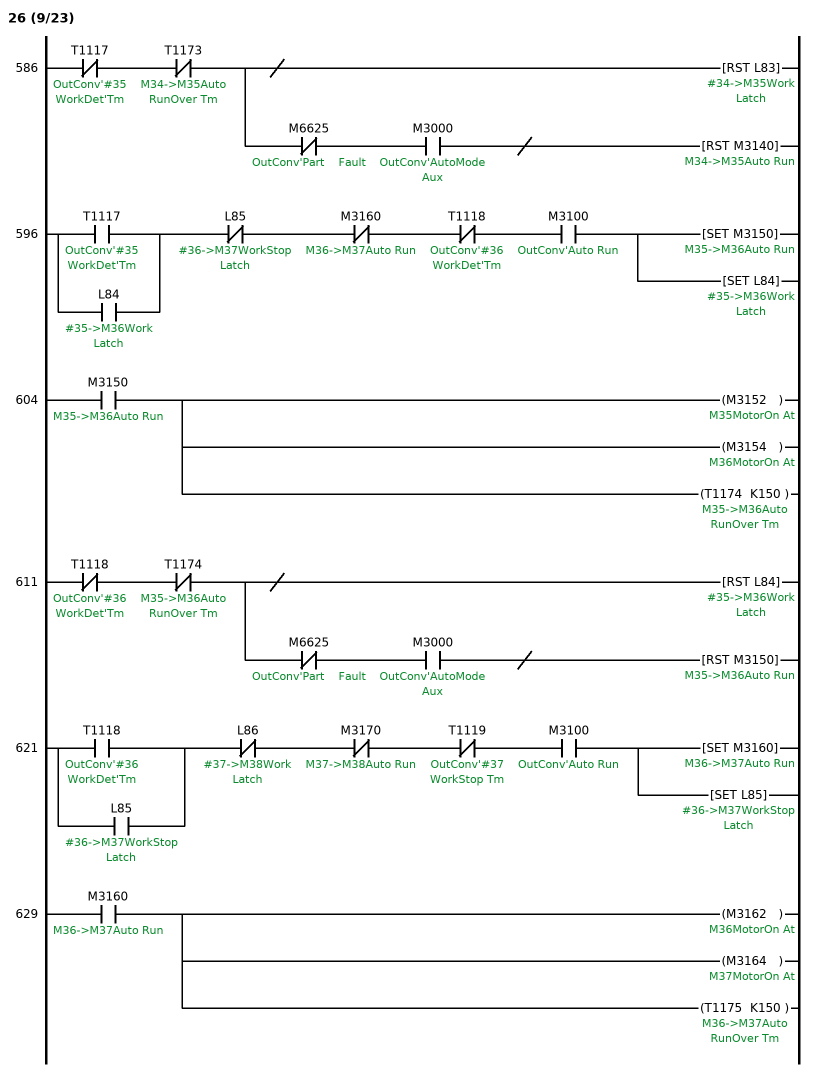
586   LDI     T1117  ; OutConv'#35 WorkDet'Tm
      ANI     T1173  ; M34->M35Auto RunOver Tm
      MPS
      INV
      RST     L83  ; #34->M35Work    Latch
      MPP
      ANI     M6625  ; OutConv'Part    Fault
      AND     M3000  ; OutConv'AutoModeAux
      INV
      RST     M3140  ; M34->M35Auto Run
596   LD      T1117  ; OutConv'#35 WorkDet'Tm
      OR      L84  ; #35->M36Work    Latch
      ANI     L85  ; #36->M37WorkStopLatch
      ANI     M3160  ; M36->M37Auto Run
      ANI     T1118  ; OutConv'#36 WorkDet'Tm
      AND     M3100  ; OutConv'Auto Run
      SET     M3150  ; M35->M36Auto Run
      SET     L84  ; #35->M36Work    Latch
604   LD      M3150  ; M35->M36Auto Run
      OUT     M3152  ; M35MotorOn At
      OUT     M3154  ; M36MotorOn At
      OUT     T1174 K150  ; M35->M36Auto RunOver Tm
611   LDI     T1118  ; OutConv'#36 WorkDet'Tm
      ANI     T1174  ; M35->M36Auto RunOver Tm
      MPS
      INV
      RST     L84  ; #35->M36Work    Latch
      MPP
      ANI     M6625  ; OutConv'Part    Fault
      AND     M3000  ; OutConv'AutoModeAux
      INV
      RST     M3150  ; M35->M36Auto Run
621   LD      T1118  ; OutConv'#36 WorkDet'Tm
      OR      L85  ; #36->M37WorkStopLatch
      ANI     L86  ; #37->M38Work    Latch
      ANI     M3170  ; M37->M38Auto Run
      ANI     T1119  ; OutConv'#37 WorkStop Tm
      AND     M3100  ; OutConv'Auto Run
      SET     M3160  ; M36->M37Auto Run
      SET     L85  ; #36->M37WorkStopLatch
629   LD      M3160  ; M36->M37Auto Run
      OUT     M3162  ; M36MotorOn At
      OUT     M3164  ; M37MotorOn At
      OUT     T1175 K150  ; M36->M37Auto RunOver Tm
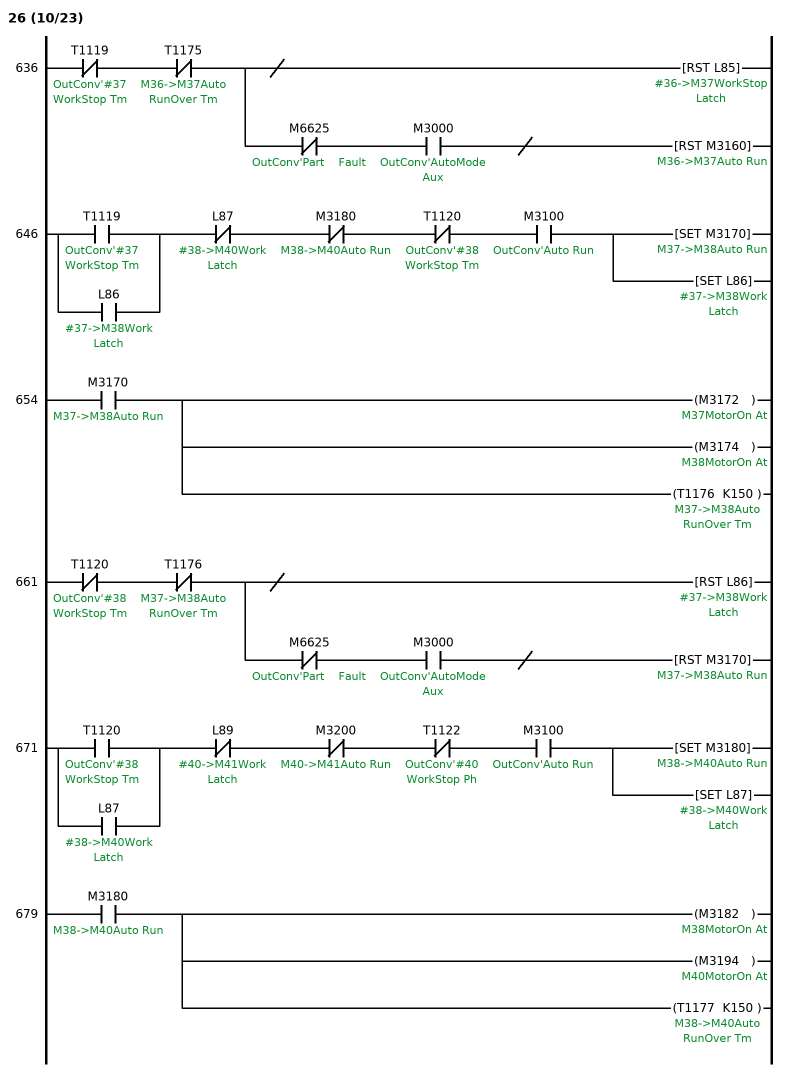
636   LDI     T1119  ; OutConv'#37 WorkStop Tm
      ANI     T1175  ; M36->M37Auto RunOver Tm
      MPS
      INV
      RST     L85  ; #36->M37WorkStopLatch
      MPP
      ANI     M6625  ; OutConv'Part    Fault
      AND     M3000  ; OutConv'AutoModeAux
      INV
      RST     M3160  ; M36->M37Auto Run
646   LD      T1119  ; OutConv'#37 WorkStop Tm
      OR      L86  ; #37->M38Work    Latch
      ANI     L87  ; #38->M40Work    Latch
      ANI     M3180  ; M38->M40Auto Run
      ANI     T1120  ; OutConv'#38 WorkStop Tm
      AND     M3100  ; OutConv'Auto Run
      SET     M3170  ; M37->M38Auto Run
      SET     L86  ; #37->M38Work    Latch
654   LD      M3170  ; M37->M38Auto Run
      OUT     M3172  ; M37MotorOn At
      OUT     M3174  ; M38MotorOn At
      OUT     T1176 K150  ; M37->M38Auto RunOver Tm
661   LDI     T1120  ; OutConv'#38 WorkStop Tm
      ANI     T1176  ; M37->M38Auto RunOver Tm
      MPS
      INV
      RST     L86  ; #37->M38Work    Latch
      MPP
      ANI     M6625  ; OutConv'Part    Fault
      AND     M3000  ; OutConv'AutoModeAux
      INV
      RST     M3170  ; M37->M38Auto Run
671   LD      T1120  ; OutConv'#38 WorkStop Tm
      OR      L87  ; #38->M40Work    Latch
      ANI     L89  ; #40->M41Work    Latch
      ANI     M3200  ; M40->M41Auto Run
      ANI     T1122  ; OutConv'#40 WorkStop Ph
      AND     M3100  ; OutConv'Auto Run
      SET     M3180  ; M38->M40Auto Run
      SET     L87  ; #38->M40Work    Latch
679   LD      M3180  ; M38->M40Auto Run
      OUT     M3182  ; M38MotorOn At
      OUT     M3194  ; M40MotorOn At
      OUT     T1177 K150  ; M38->M40Auto RunOver Tm
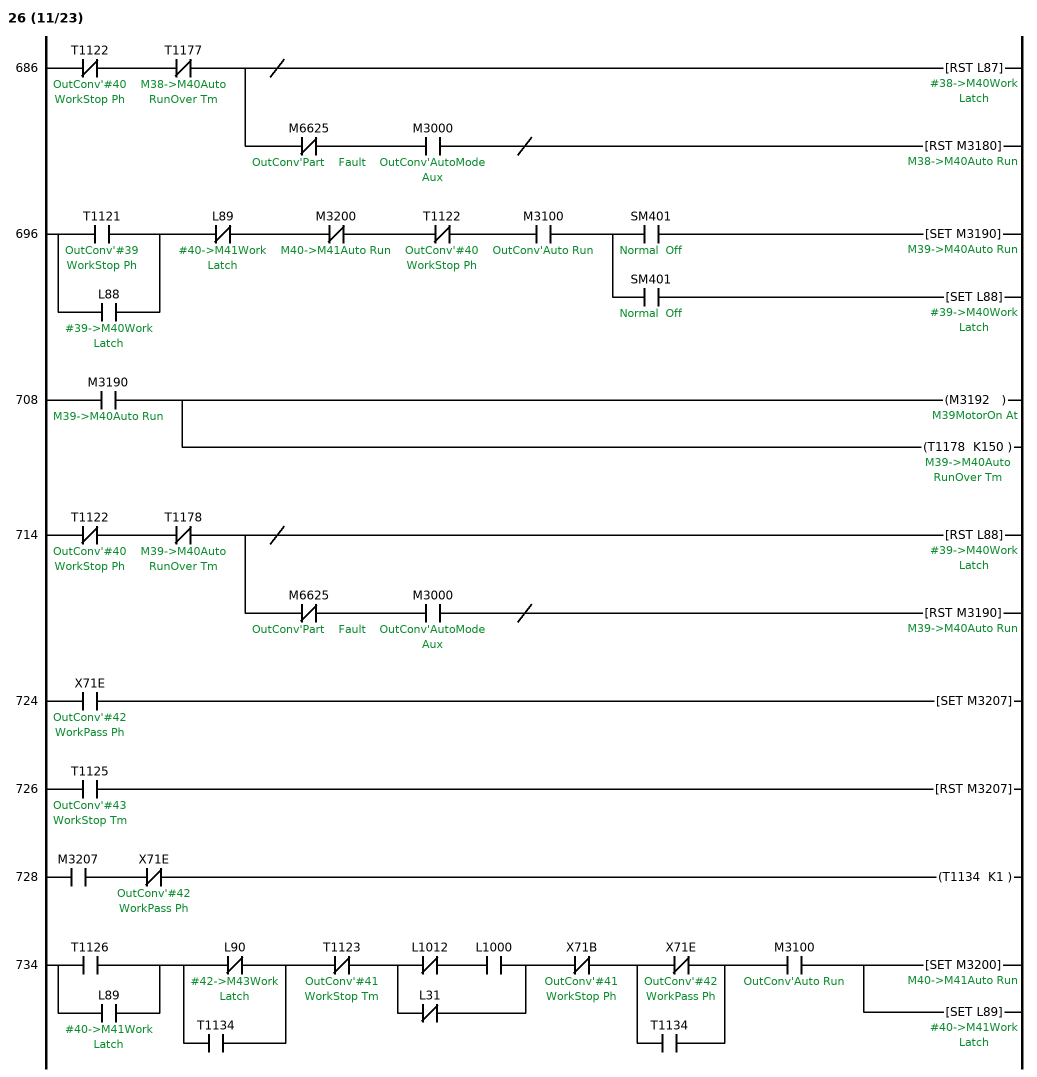
686   LDI     T1122  ; OutConv'#40 WorkStop Ph
      ANI     T1177  ; M38->M40Auto RunOver Tm
      MPS
      INV
      RST     L87  ; #38->M40Work    Latch
      MPP
      ANI     M6625  ; OutConv'Part    Fault
      AND     M3000  ; OutConv'AutoModeAux
      INV
      RST     M3180  ; M38->M40Auto Run
696   LD      T1121  ; OutConv'#39 WorkStop Ph
      OR      L88  ; #39->M40Work    Latch
      ANI     L89  ; #40->M41Work    Latch
      ANI     M3200  ; M40->M41Auto Run
      ANI     T1122  ; OutConv'#40 WorkStop Ph
      AND     M3100  ; OutConv'Auto Run
      MPS
      AND     SM401  ; Normal  Off
      SET     M3190  ; M39->M40Auto Run
      MPP
      AND     SM401  ; Normal  Off
      SET     L88  ; #39->M40Work    Latch
708   LD      M3190  ; M39->M40Auto Run
      OUT     M3192  ; M39MotorOn At
      OUT     T1178 K150  ; M39->M40Auto RunOver Tm
714   LDI     T1122  ; OutConv'#40 WorkStop Ph
      ANI     T1178  ; M39->M40Auto RunOver Tm
      MPS
      INV
      RST     L88  ; #39->M40Work    Latch
      MPP
      ANI     M6625  ; OutConv'Part    Fault
      AND     M3000  ; OutConv'AutoModeAux
      INV
      RST     M3190  ; M39->M40Auto Run
724   LD      X71E  ; OutConv'#42 WorkPass Ph
      SET     M3207
726   LD      T1125  ; OutConv'#43 WorkStop Tm
      RST     M3207
728   LD      M3207
      ANI     X71E  ; OutConv'#42 WorkPass Ph
      OUT     T1134 K1
734   LD      T1126
      OR      L89  ; #40->M41Work    Latch
      LDI     L90  ; #42->M43Work    Latch
      OR      T1134
      ANB
      ANI     T1123  ; OutConv'#41 WorkStop Tm
      LDI     L1012
      AND     L1000
      ORI     L31
      ANB
      ANI     X71B  ; OutConv'#41 WorkStop Ph
      LDI     X71E  ; OutConv'#42 WorkPass Ph
      OR      T1134
      ANB
      AND     M3100  ; OutConv'Auto Run
      SET     M3200  ; M40->M41Auto Run
      SET     L89  ; #40->M41Work    Latch
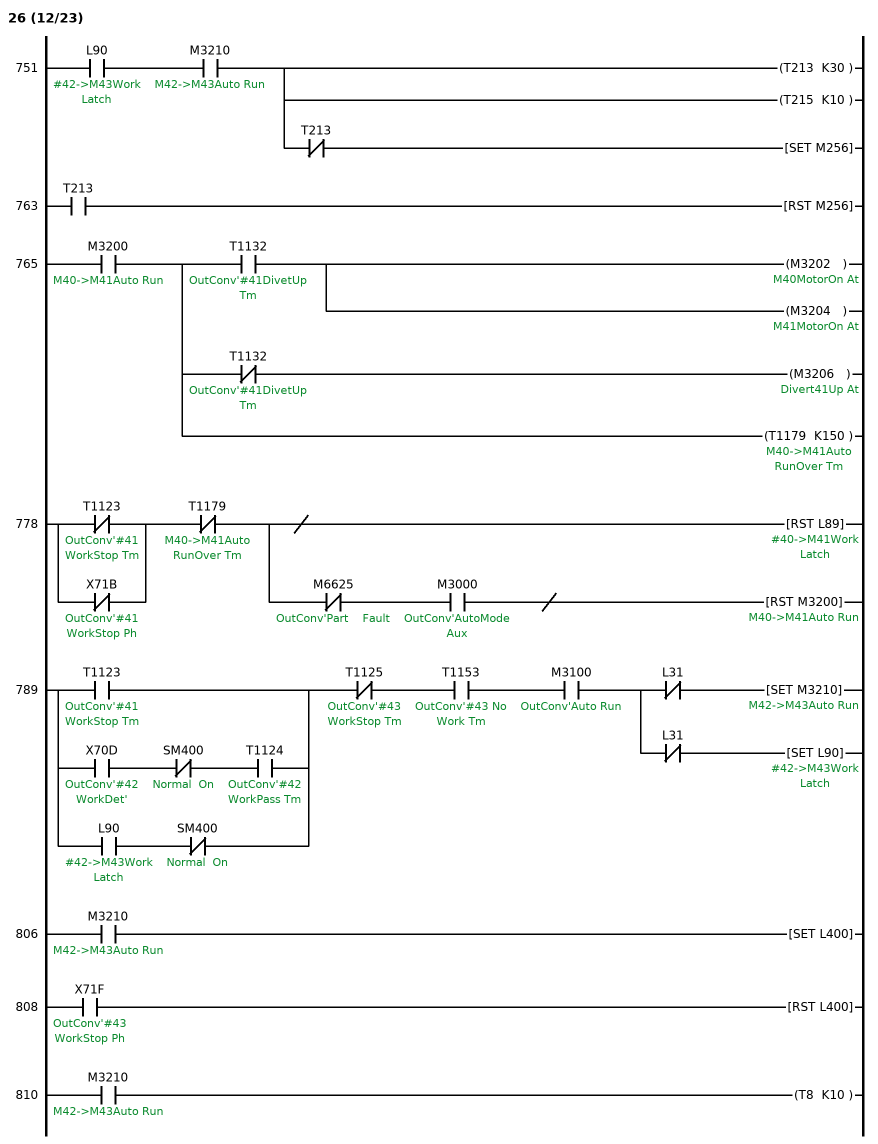
751   LD      L90  ; #42->M43Work    Latch
      AND     M3210  ; M42->M43Auto Run
      OUT     T213 K30
      OUT     T215 K10
      ANI     T213
      SET     M256
763   LD      T213
      RST     M256
765   LD      M3200  ; M40->M41Auto Run
      MPS
      AND     T1132  ; OutConv'#41DivetUp Tm
      OUT     M3202  ; M40MotorOn At
      OUT     M3204  ; M41MotorOn At
      MRD
      ANI     T1132  ; OutConv'#41DivetUp Tm
      OUT     M3206  ; Divert41Up At
      MPP
      OUT     T1179 K150  ; M40->M41Auto RunOver Tm
778   LDI     T1123  ; OutConv'#41 WorkStop Tm
      ORI     X71B  ; OutConv'#41 WorkStop Ph
      ANI     T1179  ; M40->M41Auto RunOver Tm
      MPS
      INV
      RST     L89  ; #40->M41Work    Latch
      MPP
      ANI     M6625  ; OutConv'Part    Fault
      AND     M3000  ; OutConv'AutoModeAux
      INV
      RST     M3200  ; M40->M41Auto Run
789   LD      T1123  ; OutConv'#41 WorkStop Tm
      LD      X70D  ; OutConv'#42 WorkDet'
      ANI     SM400  ; Normal  On
      AND     T1124  ; OutConv'#42 WorkPass Tm
      ORB
      LD      L90  ; #42->M43Work    Latch
      ANI     SM400  ; Normal  On
      ORB
      ANI     T1125  ; OutConv'#43 WorkStop Tm
      AND     T1153  ; OutConv'#43 No  Work Tm
      AND     M3100  ; OutConv'Auto Run
      MPS
      ANI     L31
      SET     M3210  ; M42->M43Auto Run
      MPP
      ANI     L31
      SET     L90  ; #42->M43Work    Latch
806   LD      M3210  ; M42->M43Auto Run
      SET     L400
808   LD      X71F  ; OutConv'#43 WorkStop Ph
      RST     L400
810   LD      M3210  ; M42->M43Auto Run
      OUT     T8 K10
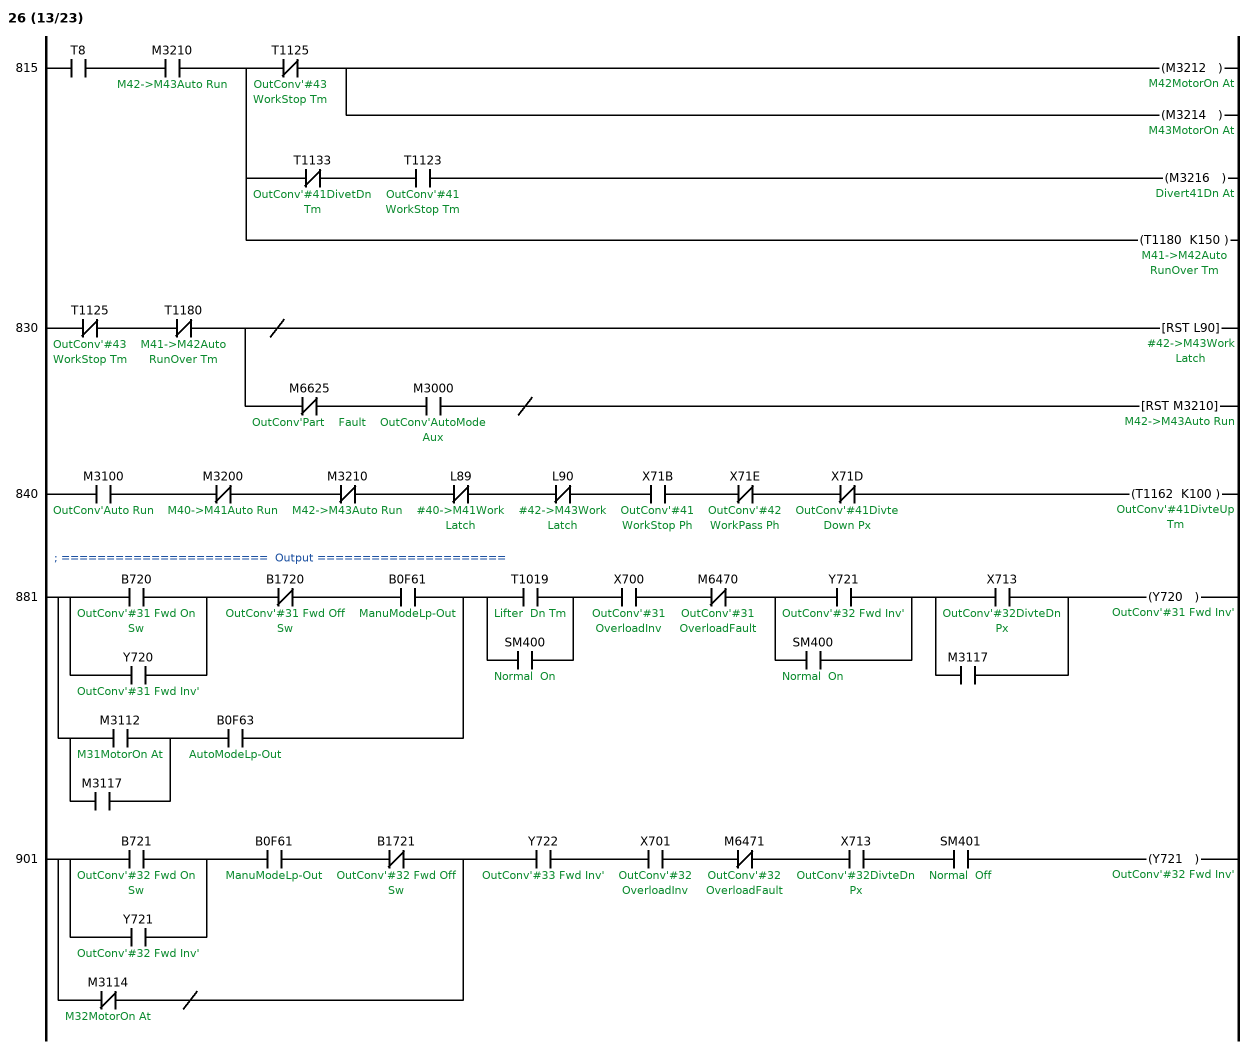
815   LD      T8
      AND     M3210  ; M42->M43Auto Run
      MPS
      ANI     T1125  ; OutConv'#43 WorkStop Tm
      OUT     M3212  ; M42MotorOn At
      OUT     M3214  ; M43MotorOn At
      MRD
      ANI     T1133  ; OutConv'#41DivetDn Tm
      AND     T1123  ; OutConv'#41 WorkStop Tm
      OUT     M3216  ; Divert41Dn At
      MPP
      OUT     T1180 K150  ; M41->M42Auto RunOver Tm
830   LDI     T1125  ; OutConv'#43 WorkStop Tm
      ANI     T1180  ; M41->M42Auto RunOver Tm
      MPS
      INV
      RST     L90  ; #42->M43Work    Latch
      MPP
      ANI     M6625  ; OutConv'Part    Fault
      AND     M3000  ; OutConv'AutoModeAux
      INV
      RST     M3210  ; M42->M43Auto Run
840   LD      M3100  ; OutConv'Auto Run
      ANI     M3200  ; M40->M41Auto Run
      ANI     M3210  ; M42->M43Auto Run
      ANI     L89  ; #40->M41Work    Latch
      ANI     L90  ; #42->M43Work    Latch
      AND     X71B  ; OutConv'#41 WorkStop Ph
      ANI     X71E  ; OutConv'#42 WorkPass Ph
      ANI     X71D  ; OutConv'#41DivteDown Px
      OUT     T1162 K100  ; OutConv'#41DivteUp Tm
; =======================  Output =====================
881   LD      B720  ; OutConv'#31 Fwd On Sw
      OR      Y720  ; OutConv'#31 Fwd Inv'
      ANI     B1720  ; OutConv'#31 Fwd Off Sw
      AND     B0F61  ; ManuModeLp-Out
      LD      M3112  ; M31MotorOn At
      OR      M3117
      AND     B0F63  ; AutoModeLp-Out
      ORB
      LD      T1019  ; Lifter  Dn Tm
      OR      SM400  ; Normal  On
      ANB
      AND     X700  ; OutConv'#31     OverloadInv
      ANI     M6470  ; OutConv'#31     OverloadFault
      LD      Y721  ; OutConv'#32 Fwd Inv'
      OR      SM400  ; Normal  On
      ANB
      LD      X713  ; OutConv'#32DivteDn Px
      OR      M3117
      ANB
      OUT     Y720  ; OutConv'#31 Fwd Inv'
901   LD      B721  ; OutConv'#32 Fwd On Sw
      OR      Y721  ; OutConv'#32 Fwd Inv'
      AND     B0F61  ; ManuModeLp-Out
      ANI     B1721  ; OutConv'#32 Fwd Off Sw
      LDI     M3114  ; M32MotorOn At
      INV
      ORB
      AND     Y722  ; OutConv'#33 Fwd Inv'
      AND     X701  ; OutConv'#32     OverloadInv
      ANI     M6471  ; OutConv'#32     OverloadFault
      AND     X713  ; OutConv'#32DivteDn Px
      AND     SM401  ; Normal  Off
      OUT     Y721  ; OutConv'#32 Fwd Inv'
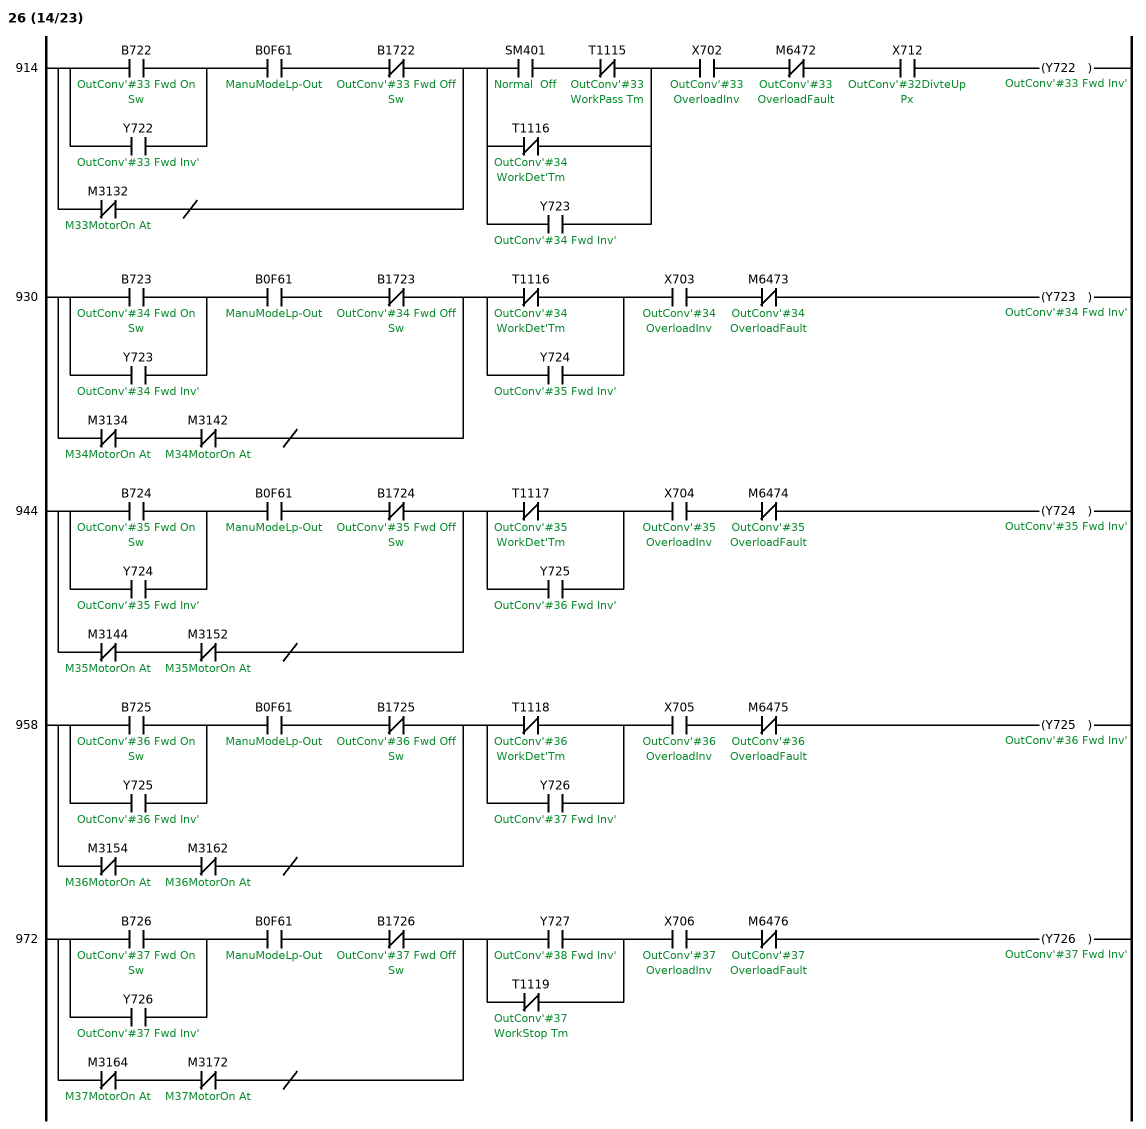
914   LD      B722  ; OutConv'#33 Fwd On Sw
      OR      Y722  ; OutConv'#33 Fwd Inv'
      AND     B0F61  ; ManuModeLp-Out
      ANI     B1722  ; OutConv'#33 Fwd Off Sw
      LDI     M3132  ; M33MotorOn At
      INV
      ORB
      LD      SM401  ; Normal  Off
      ANI     T1115  ; OutConv'#33 WorkPass Tm
      ORI     T1116  ; OutConv'#34 WorkDet'Tm
      OR      Y723  ; OutConv'#34 Fwd Inv'
      ANB
      AND     X702  ; OutConv'#33     OverloadInv
      ANI     M6472  ; OutConv'#33     OverloadFault
      AND     X712  ; OutConv'#32DivteUp Px
      OUT     Y722  ; OutConv'#33 Fwd Inv'
930   LD      B723  ; OutConv'#34 Fwd On Sw
      OR      Y723  ; OutConv'#34 Fwd Inv'
      AND     B0F61  ; ManuModeLp-Out
      ANI     B1723  ; OutConv'#34 Fwd Off Sw
      LDI     M3134  ; M34MotorOn At
      ANI     M3142  ; M34MotorOn At
      INV
      ORB
      LDI     T1116  ; OutConv'#34 WorkDet'Tm
      OR      Y724  ; OutConv'#35 Fwd Inv'
      ANB
      AND     X703  ; OutConv'#34     OverloadInv
      ANI     M6473  ; OutConv'#34     OverloadFault
      OUT     Y723  ; OutConv'#34 Fwd Inv'
944   LD      B724  ; OutConv'#35 Fwd On Sw
      OR      Y724  ; OutConv'#35 Fwd Inv'
      AND     B0F61  ; ManuModeLp-Out
      ANI     B1724  ; OutConv'#35 Fwd Off Sw
      LDI     M3144  ; M35MotorOn At
      ANI     M3152  ; M35MotorOn At
      INV
      ORB
      LDI     T1117  ; OutConv'#35 WorkDet'Tm
      OR      Y725  ; OutConv'#36 Fwd Inv'
      ANB
      AND     X704  ; OutConv'#35     OverloadInv
      ANI     M6474  ; OutConv'#35     OverloadFault
      OUT     Y724  ; OutConv'#35 Fwd Inv'
958   LD      B725  ; OutConv'#36 Fwd On Sw
      OR      Y725  ; OutConv'#36 Fwd Inv'
      AND     B0F61  ; ManuModeLp-Out
      ANI     B1725  ; OutConv'#36 Fwd Off Sw
      LDI     M3154  ; M36MotorOn At
      ANI     M3162  ; M36MotorOn At
      INV
      ORB
      LDI     T1118  ; OutConv'#36 WorkDet'Tm
      OR      Y726  ; OutConv'#37 Fwd Inv'
      ANB
      AND     X705  ; OutConv'#36     OverloadInv
      ANI     M6475  ; OutConv'#36     OverloadFault
      OUT     Y725  ; OutConv'#36 Fwd Inv'
972   LD      B726  ; OutConv'#37 Fwd On Sw
      OR      Y726  ; OutConv'#37 Fwd Inv'
      AND     B0F61  ; ManuModeLp-Out
      ANI     B1726  ; OutConv'#37 Fwd Off Sw
      LDI     M3164  ; M37MotorOn At
      ANI     M3172  ; M37MotorOn At
      INV
      ORB
      LD      Y727  ; OutConv'#38 Fwd Inv'
      ORI     T1119  ; OutConv'#37 WorkStop Tm
      ANB
      AND     X706  ; OutConv'#37     OverloadInv
      ANI     M6476  ; OutConv'#37     OverloadFault
      OUT     Y726  ; OutConv'#37 Fwd Inv'
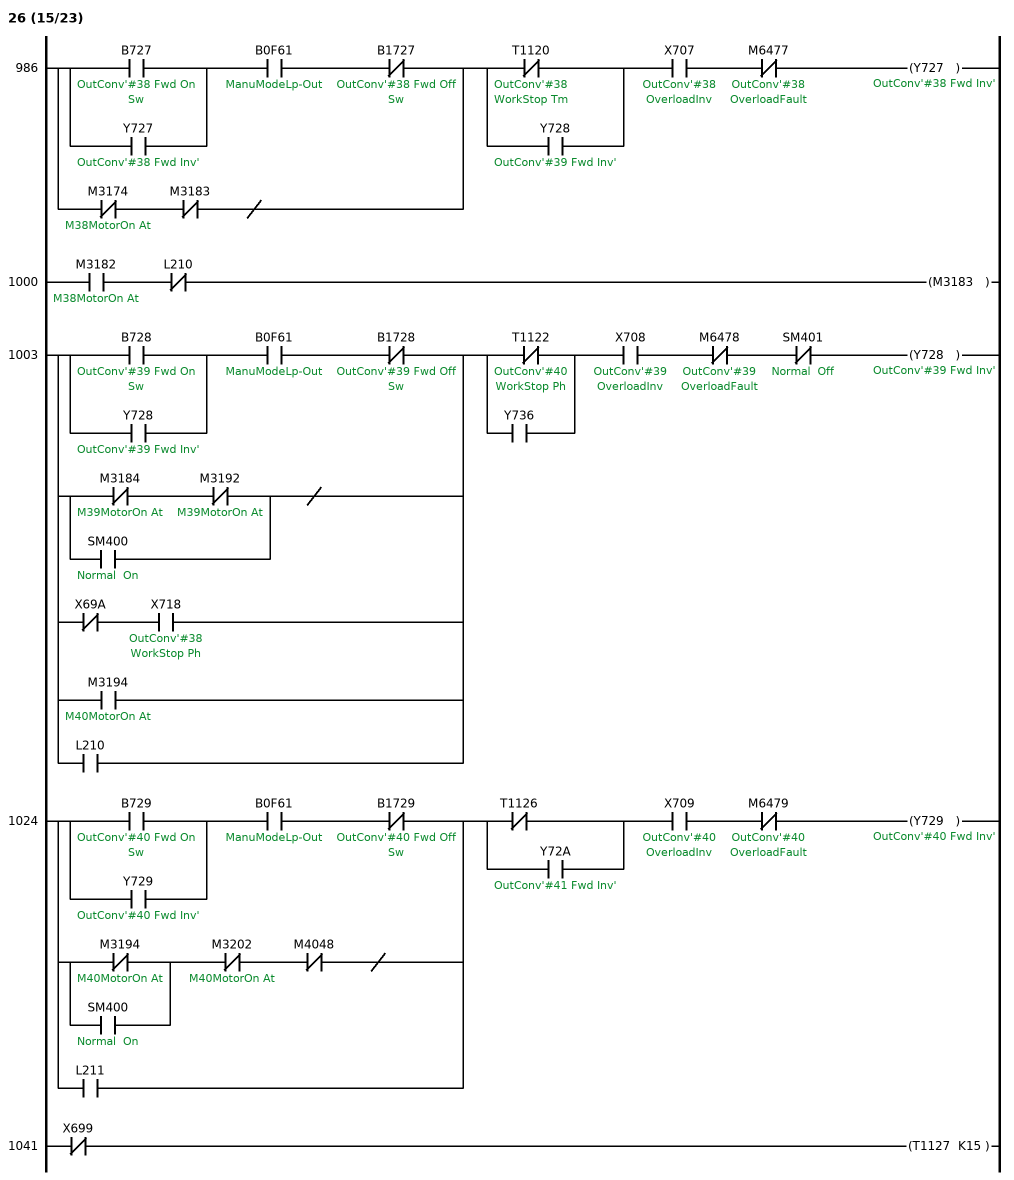
986   LD      B727  ; OutConv'#38 Fwd On Sw
      OR      Y727  ; OutConv'#38 Fwd Inv'
      AND     B0F61  ; ManuModeLp-Out
      ANI     B1727  ; OutConv'#38 Fwd Off Sw
      LDI     M3174  ; M38MotorOn At
      ANI     M3183
      INV
      ORB
      LDI     T1120  ; OutConv'#38 WorkStop Tm
      OR      Y728  ; OutConv'#39 Fwd Inv'
      ANB
      AND     X707  ; OutConv'#38     OverloadInv
      ANI     M6477  ; OutConv'#38     OverloadFault
      OUT     Y727  ; OutConv'#38 Fwd Inv'
1000  LD      M3182  ; M38MotorOn At
      ANI     L210
      OUT     M3183
1003  LD      B728  ; OutConv'#39 Fwd On Sw
      OR      Y728  ; OutConv'#39 Fwd Inv'
      AND     B0F61  ; ManuModeLp-Out
      ANI     B1728  ; OutConv'#39 Fwd Off Sw
      LDI     M3184  ; M39MotorOn At
      ANI     M3192  ; M39MotorOn At
      OR      SM400  ; Normal  On
      INV
      ORB
      LDI     X69A
      AND     X718  ; OutConv'#38 WorkStop Ph
      ORB
      OR      M3194  ; M40MotorOn At
      OR      L210
      LDI     T1122  ; OutConv'#40 WorkStop Ph
      OR      Y736
      ANB
      AND     X708  ; OutConv'#39     OverloadInv
      ANI     M6478  ; OutConv'#39     OverloadFault
      ANI     SM401  ; Normal  Off
      OUT     Y728  ; OutConv'#39 Fwd Inv'
1024  LD      B729  ; OutConv'#40 Fwd On Sw
      OR      Y729  ; OutConv'#40 Fwd Inv'
      AND     B0F61  ; ManuModeLp-Out
      ANI     B1729  ; OutConv'#40 Fwd Off Sw
      LDI     M3194  ; M40MotorOn At
      OR      SM400  ; Normal  On
      ANI     M3202  ; M40MotorOn At
      ANI     M4048
      INV
      ORB
      OR      L211
      LDI     T1126
      OR      Y72A  ; OutConv'#41 Fwd Inv'
      ANB
      AND     X709  ; OutConv'#40     OverloadInv
      ANI     M6479  ; OutConv'#40     OverloadFault
      OUT     Y729  ; OutConv'#40 Fwd Inv'
1041  LDI     X699
      OUT     T1127 K15
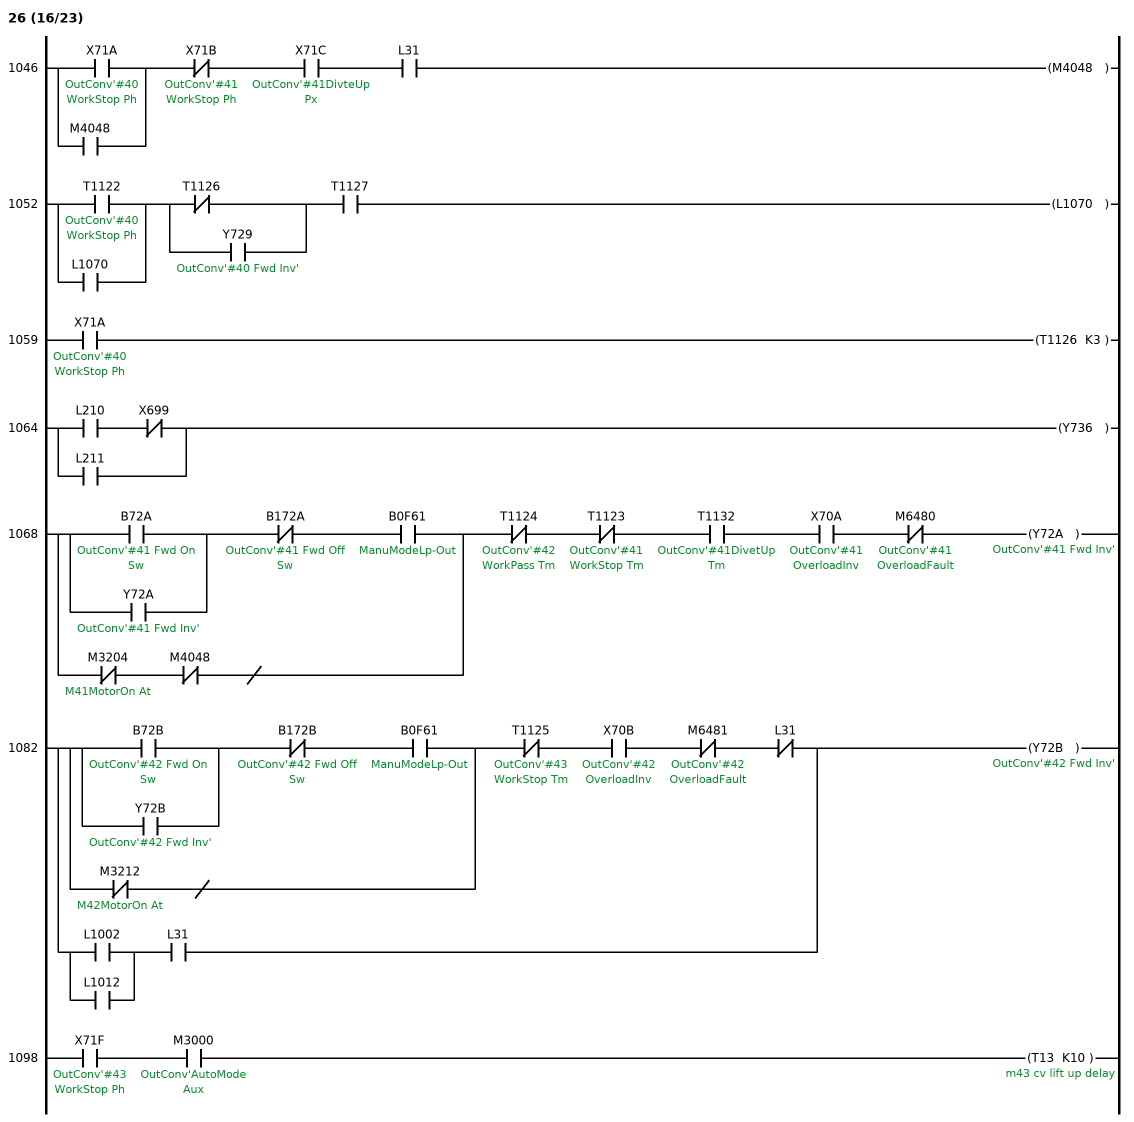
1046  LD      X71A  ; OutConv'#40 WorkStop Ph
      OR      M4048
      ANI     X71B  ; OutConv'#41 WorkStop Ph
      AND     X71C  ; OutConv'#41DivteUp Px
      AND     L31
      OUT     M4048
1052  LD      T1122  ; OutConv'#40 WorkStop Ph
      OR      L1070
      LDI     T1126
      OR      Y729  ; OutConv'#40 Fwd Inv'
      ANB
      AND     T1127
      OUT     L1070
1059  LD      X71A  ; OutConv'#40 WorkStop Ph
      OUT     T1126 K3
1064  LD      L210
      ANI     X699
      OR      L211
      OUT     Y736
1068  LD      B72A  ; OutConv'#41 Fwd On Sw
      OR      Y72A  ; OutConv'#41 Fwd Inv'
      ANI     B172A  ; OutConv'#41 Fwd Off Sw
      AND     B0F61  ; ManuModeLp-Out
      LDI     M3204  ; M41MotorOn At
      ANI     M4048
      INV
      ORB
      ANI     T1124  ; OutConv'#42 WorkPass Tm
      ANI     T1123  ; OutConv'#41 WorkStop Tm
      AND     T1132  ; OutConv'#41DivetUp Tm
      AND     X70A  ; OutConv'#41     OverloadInv
      ANI     M6480  ; OutConv'#41     OverloadFault
      OUT     Y72A  ; OutConv'#41 Fwd Inv'
1082  LD      B72B  ; OutConv'#42 Fwd On Sw
      OR      Y72B  ; OutConv'#42 Fwd Inv'
      ANI     B172B  ; OutConv'#42 Fwd Off Sw
      AND     B0F61  ; ManuModeLp-Out
      LDI     M3212  ; M42MotorOn At
      INV
      ORB
      ANI     T1125  ; OutConv'#43 WorkStop Tm
      AND     X70B  ; OutConv'#42     OverloadInv
      ANI     M6481  ; OutConv'#42     OverloadFault
      ANI     L31
      LD      L1002
      OR      L1012
      AND     L31
      ORB
      OUT     Y72B  ; OutConv'#42 Fwd Inv'
1098  LD      X71F  ; OutConv'#43 WorkStop Ph
      AND     M3000  ; OutConv'AutoModeAux
      OUT     T13 K10  ; m43 cv lift up delay
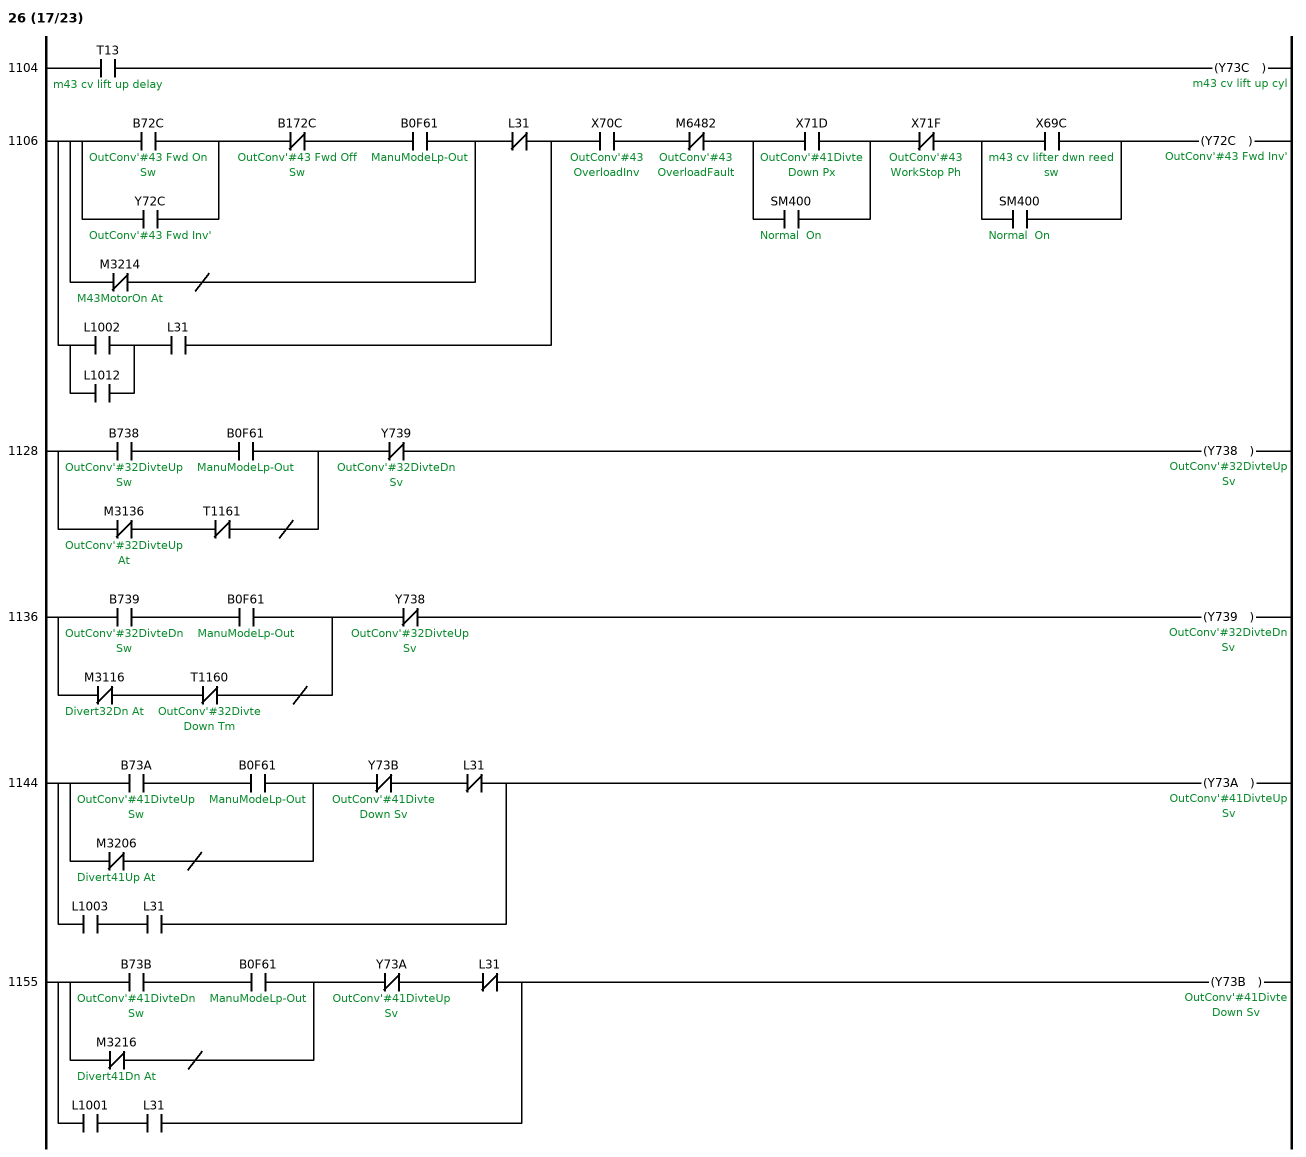
1104  LD      T13  ; m43 cv lift up delay
      OUT     Y73C  ; m43 cv lift up cyl
1106  LD      B72C  ; OutConv'#43 Fwd On Sw
      OR      Y72C  ; OutConv'#43 Fwd Inv'
      ANI     B172C  ; OutConv'#43 Fwd Off Sw
      AND     B0F61  ; ManuModeLp-Out
      LDI     M3214  ; M43MotorOn At
      INV
      ORB
      ANI     L31
      LD      L1002
      OR      L1012
      AND     L31
      ORB
      AND     X70C  ; OutConv'#43     OverloadInv
      ANI     M6482  ; OutConv'#43     OverloadFault
      LD      X71D  ; OutConv'#41DivteDown Px
      OR      SM400  ; Normal  On
      ANB
      ANI     X71F  ; OutConv'#43 WorkStop Ph
      LD      X69C  ; m43 cv lifter dwn reed sw
      OR      SM400  ; Normal  On
      ANB
      OUT     Y72C  ; OutConv'#43 Fwd Inv'
1128  LD      B738  ; OutConv'#32DivteUp Sw
      AND     B0F61  ; ManuModeLp-Out
      LDI     M3136  ; OutConv'#32DivteUp At
      ANI     T1161
      INV
      ORB
      ANI     Y739  ; OutConv'#32DivteDn Sv
      OUT     Y738  ; OutConv'#32DivteUp Sv
1136  LD      B739  ; OutConv'#32DivteDn Sw
      AND     B0F61  ; ManuModeLp-Out
      LDI     M3116  ; Divert32Dn At
      ANI     T1160  ; OutConv'#32DivteDown Tm
      INV
      ORB
      ANI     Y738  ; OutConv'#32DivteUp Sv
      OUT     Y739  ; OutConv'#32DivteDn Sv
1144  LD      B73A  ; OutConv'#41DivteUp Sw
      AND     B0F61  ; ManuModeLp-Out
      LDI     M3206  ; Divert41Up At
      INV
      ORB
      ANI     Y73B  ; OutConv'#41DivteDown Sv
      ANI     L31
      LD      L1003
      AND     L31
      ORB
      OUT     Y73A  ; OutConv'#41DivteUp Sv
1155  LD      B73B  ; OutConv'#41DivteDn Sw
      AND     B0F61  ; ManuModeLp-Out
      LDI     M3216  ; Divert41Dn At
      INV
      ORB
      ANI     Y73A  ; OutConv'#41DivteUp Sv
      ANI     L31
      LD      L1001
      AND     L31
      ORB
      OUT     Y73B  ; OutConv'#41DivteDown Sv
